LIN {X 0,Y 419.914,Z 1009.254,A -85,B 0,C 180,E1 17766.267,E2 17766.267} C_VEL
LIN {X 0,Y 411.556,Z 1028.718,A -85,B 0,C 180,E1 17763.636,E2 17763.636} C_VEL
LIN {X 0,Y 404.819,Z 1043.815,A -85,B 0,C 180,E1 17761.243,E2 17761.243} C_VEL
LIN {X 0,Y 398.369,Z 1058.063,A -85,B 0,C 180,E1 17758.645,E2 17758.645} C_VEL
LIN {X 0,Y 391.155,Z 1073.748,A -85,B 0,C 180,E1 17755.27,E2 17755.27} C_VEL
LIN {X 0,Y 385.875,Z 1085.364,A -85,B 0,C 180,E1 17752.321,E2 17752.321} C_VEL
LIN {X 0,Y 380.976,Z 1096.633,A -85,B 0,C 180,E1 17748.992,E2 17748.992} C_VEL
LIN {X 0,Y 376.618,Z 1107.153,A -85,B 0,C 180,E1 17745.238,E2 17745.238} C_VEL
LIN {X 0,Y 373.797,Z 1114.641,A -85,B 0,C 180,E1 17742.043,E2 17742.043} C_VEL
LIN {X 0,Y 371.603,Z 1121.269,A -85,B 0,C 180,E1 17738.666,E2 17738.666} C_VEL
LIN {X 0,Y 369.854,Z 1127.751,A -85,B 0,C 180,E1 17734.496,E2 17734.496} C_VEL
LIN {X 0,Y 368.993,Z 1131.833,A -85,B 0,C 180,E1 17730.931,E2 17730.931} C_VEL
LIN {X 0,Y 368.608,Z 1134.428,A -85,B 0,C 180,E1 17727.824,E2 17727.824} C_VEL
LIN {X 0,Y 368.429,Z 1136.13,A -85,B 0,C 180,E1 17724.706,E2 17724.706} C_VEL
LIN {X 0,Y 368.395,Z 1136.967,A -85,B 0,C 180,E1 17721.415,E2 17721.415} C_VEL
LIN {X 0,Y 368.477,Z 1136.697,A -85,B 0,C 180,E1 17717.415,E2 17717.415} C_VEL
LIN {X 0,Y 367.526,Z 1136.369,A -85,B 0,C 180,E1 17716.218,E2 17716.218} C_VEL
LIN {X 0,Y 361.39,Z 1135.259,A -85,B 0,C 180,E1 17712.831,E2 17712.831} C_VEL
LIN {X 0,Y 360.995,Z 1134.749,A -85,B 0,C 180,E1 17711.95,E2 17711.95} C_VEL
LIN {X 0,Y 362,Z 1130.889,A -85,B 0,C 180,E1 17707.716,E2 17707.716} C_VEL
LIN {X 0,Y 363.474,Z 1126.513,A -85,B 0,C 180,E1 17704.238,E2 17704.238} C_VEL
LIN {X 0,Y 365.707,Z 1120.907,A -85,B 0,C 180,E1 17700.699,E2 17700.699} C_VEL
LIN {X 0,Y 369.605,Z 1112.44,A -85,B 0,C 180,E1 17696.432,E2 17696.432} C_VEL
LIN {X 0,Y 374.095,Z 1103.44,A -85,B 0,C 180,E1 17692.798,E2 17692.798} C_VEL
LIN {X 0,Y 379.173,Z 1093.949,A -85,B 0,C 180,E1 17689.557,E2 17689.557} C_VEL
LIN {X 0,Y 386.62,Z 1080.458,A -85,B 0,C 180,E1 17685.712,E2 17685.712} C_VEL
LIN {X 0,Y 393.537,Z 1068.018,A -85,B 0,C 180,E1 17682.755,E2 17682.755} C_VEL
LIN {X 0,Y 400.925,Z 1054.718,A -85,B 0,C 180,E1 17680.038,E2 17680.038} C_VEL
LIN {X 0,Y 410.659,Z 1036.667,A -85,B 0,C 180,E1 17676.93,E2 17676.93} C_VEL
LIN {X 0,Y 418.509,Z 1021.522,A -85,B 0,C 180,E1 17674.73,E2 17674.73} C_VEL
LIN {X 0,Y 426.535,Z 1005.366,A -85,B 0,C 180,E1 17672.696,E2 17672.696} C_VEL
LIN {X 0,Y 436.473,Z 984.02,A -85,B 0,C 180,E1 17670.416,E2 17670.416} C_VEL
LIN {X 0,Y 444.603,Z 964.996,A -85,B 0,C 180,E1 17668.71,E2 17668.71} C_VEL
LIN {X 0,Y 451.802,Z 946.841,A -85,B 0,C 180,E1 17667.31,E2 17667.31} C_VEL
LIN {X 0,Y 459.9,Z 924.448,A -85,B 0,C 180,E1 17665.833,E2 17665.833} C_VEL
LIN {X 0,Y 466.882,Z 902.195,A -85,B 0,C 180,E1 17664.619,E2 17664.619} C_VEL
LIN {X 0,Y 472.272,Z 882.801,A -85,B 0,C 180,E1 17663.72,E2 17663.72} C_VEL
LIN {X 0,Y 477.499,Z 861.186,A -85,B 0,C 180,E1 17662.878,E2 17662.878} C_VEL
LIN {X 0,Y 483.038,Z 832.99,A -85,B 0,C 180,E1 17662.009,E2 17662.009} C_VEL
LIN {X 0,Y 486.435,Z 810.58,A -85,B 0,C 180,E1 17661.488,E2 17661.488} C_VEL
LIN {X 0,Y 488.932,Z 787.935,A -85,B 0,C 180,E1 17661.074,E2 17661.074} C_VEL
LIN {X 0,Y 507.571,Z 549.143,A -85,B 0,C 180,E1 17657.399,E2 17657.399} C_VEL
LIN {X 0,Y 510.985,Z 506.859,A -85,B 0,C 180,E1 17656.756,E2 17656.756} C_VEL
LIN {X 0,Y 505.744,Z 497.944,A -85,B 0,C 180,E1 17654.6,E2 17654.6} C_VEL
LIN {X 0,Y 500.413,Z 489.376,A -85,B 0,C 180,E1 17652.052,E2 17652.052} C_VEL
LIN {X 0,Y 497.211,Z 484.357,A -85,B 0,C 180,E1 17650.252,E2 17650.252} C_VEL
LIN {X 0,Y 494.031,Z 479.444,A -85,B 0,C 180,E1 17648.145,E2 17648.145} C_VEL
LIN {X 0,Y 492.423,Z 477.013,A -85,B 0,C 180,E1 17646.881,E2 17646.881} C_VEL
LIN {X 0,Y 489.648,Z 472.649,A -85,B 0,C 180,E1 17644.099,E2 17644.099} C_VEL
LIN {X 0,Y 487.171,Z 469.067,A -85,B 0,C 180,E1 17638.942,E2 17638.942} C_VEL
LIN {X 0,Y 487.223,Z 469.186,A -85,B 0,C 180,E1 17636.47,E2 17636.47} C_VEL
LIN {X 0,Y 490.053,Z 473.176,A -85,B 0,C 180,E1 17631.138,E2 17631.138} C_VEL
LIN {X 0,Y 493.646,Z 478.878,A -85,B 0,C 180,E1 17627.839,E2 17627.839} C_VEL
LIN {X 0,Y 496.917,Z 484.03,A -85,B 0,C 180,E1 17625.611,E2 17625.611} C_VEL
LIN {X 0,Y 499.764,Z 488.535,A -85,B 0,C 180,E1 17623.972,E2 17623.972} C_VEL
LIN {X 0,Y 504.407,Z 495.808,A -85,B 0,C 180,E1 17621.688,E2 17621.688} C_VEL
LIN {X 0,Y 510.711,Z 506.476,A -85,B 0,C 180,E1 17619.038,E2 17619.038} C_VEL
LIN {X 0,Y 512.388,Z 509.7,A -85,B 0,C 180,E1 17618.385,E2 17618.385} C_VEL
LIN {X 0,Y 495.256,Z 729.15,A -85,B 0,C 180,E1 17614.92,E2 17614.92} C_VEL
LIN {X 0,Y 488.537,Z 815.817,A -85,B 0,C 180,E1 17613.529,E2 17613.529} C_VEL
LIN {X 0,Y 484.757,Z 844.781,A -85,B 0,C 180,E1 17612.964,E2 17612.964} C_VEL
LIN {X 0,Y 480.382,Z 868.6,A -85,B 0,C 180,E1 17612.377,E2 17612.377} C_VEL
LIN {X 0,Y 475.726,Z 889.877,A -85,B 0,C 180,E1 17611.719,E2 17611.719} C_VEL
LIN {X 0,Y 470.261,Z 911.48,A -85,B 0,C 180,E1 17610.91,E2 17610.91} C_VEL
LIN {X 0,Y 462.298,Z 938.776,A -85,B 0,C 180,E1 17609.65,E2 17609.65} C_VEL
LIN {X 0,Y 455.227,Z 960.106,A -85,B 0,C 180,E1 17608.452,E2 17608.452} C_VEL
LIN {X 0,Y 448.224,Z 979.553,A -85,B 0,C 180,E1 17607.174,E2 17607.174} C_VEL
LIN {X 0,Y 440.915,Z 998.4,A -85,B 0,C 180,E1 17605.748,E2 17605.748} C_VEL
LIN {X 0,Y 431.52,Z 1021.146,A -85,B 0,C 180,E1 17603.74,E2 17603.74} C_VEL
LIN {X 0,Y 422.386,Z 1041.626,A -85,B 0,C 180,E1 17601.585,E2 17601.585} C_VEL
LIN {X 0,Y 414.68,Z 1058.316,A -85,B 0,C 180,E1 17599.562,E2 17599.562} C_VEL
LIN {X 0,Y 406.899,Z 1074.752,A -85,B 0,C 180,E1 17597.284,E2 17597.284} C_VEL
LIN {X 0,Y 397.906,Z 1093.613,A -85,B 0,C 180,E1 17594.26,E2 17594.26} C_VEL
LIN {X 0,Y 389.649,Z 1110.63,A -85,B 0,C 180,E1 17591.023,E2 17591.023} C_VEL
LIN {X 0,Y 383.486,Z 1123.697,A -85,B 0,C 180,E1 17588.165,E2 17588.165} C_VEL
LIN {X 0,Y 377.582,Z 1136.795,A -85,B 0,C 180,E1 17584.888,E2 17584.888} C_VEL
LIN {X 0,Y 371.414,Z 1151.399,A -85,B 0,C 180,E1 17580.584,E2 17580.584} C_VEL
LIN {X 0,Y 367.703,Z 1161.191,A -85,B 0,C 180,E1 17577.183,E2 17577.183} C_VEL
LIN {X 0,Y 364.983,Z 1169.338,A -85,B 0,C 180,E1 17573.919,E2 17573.919} C_VEL
LIN {X 0,Y 362.911,Z 1176.713,A -85,B 0,C 180,E1 17570.481,E2 17570.481} C_VEL
LIN {X 0,Y 361.4,Z 1183.466,A -85,B 0,C 180,E1 17566.722,E2 17566.722} C_VEL
LIN {X 0,Y 360.514,Z 1189.451,A -85,B 0,C 180,E1 17562.493,E2 17562.493} C_VEL
LIN {X 0,Y 360.23,Z 1193.242,A -85,B 0,C 180,E1 17558.781,E2 17558.781} C_VEL
LIN {X 0,Y 360.196,Z 1195.573,A -85,B 0,C 180,E1 17555.416,E2 17555.416} C_VEL
LIN {X 0,Y 360.224,Z 1196.781,A -85,B 0,C 180,E1 17552.183,E2 17552.183} C_VEL
LIN {X 0,Y 360.227,Z 1196.963,A -85,B 0,C 180,E1 17549.046,E2 17549.046} C_VEL
LIN {X 0,Y 360.202,Z 1196.137,A -85,B 0,C 180,E1 17545.861,E2 17545.861} C_VEL
LIN {X 0,Y 360.215,Z 1194.293,A -85,B 0,C 180,E1 17542.664,E2 17542.664} C_VEL
LIN {X 0,Y 360.335,Z 1191.418,A -85,B 0,C 180,E1 17539.448,E2 17539.448} C_VEL
LIN {X 0,Y 360.729,Z 1187.502,A -85,B 0,C 180,E1 17536.21,E2 17536.21} C_VEL
LIN {X 0,Y 361.455,Z 1182.799,A -85,B 0,C 180,E1 17533.115,E2 17533.115} C_VEL
LIN {X 0,Y 362.753,Z 1176.781,A -85,B 0,C 180,E1 17529.847,E2 17529.847} C_VEL
LIN {X 0,Y 364.616,Z 1169.625,A -85,B 0,C 180,E1 17526.571,E2 17526.571} C_VEL
LIN {X 0,Y 367.345,Z 1160.858,A -85,B 0,C 180,E1 17523.139,E2 17523.139} C_VEL
LIN {X 0,Y 371.889,Z 1148.059,A -85,B 0,C 180,E1 17518.922,E2 17518.922} C_VEL
LIN {X 0,Y 376.613,Z 1135.964,A -85,B 0,C 180,E1 17515.564,E2 17515.564} C_VEL
LIN {X 0,Y 381.398,Z 1124.305,A -85,B 0,C 180,E1 17512.73,E2 17512.73} C_VEL
LIN {X 0,Y 387.036,Z 1110.995,A -85,B 0,C 180,E1 17509.881,E2 17509.881} C_VEL
LIN {X 0,Y 394.625,Z 1093.507,A -85,B 0,C 180,E1 17506.636,E2 17506.636} C_VEL
LIN {X 0,Y 402.156,Z 1075.877,A -85,B 0,C 180,E1 17503.862,E2 17503.862} C_VEL
LIN {X 0,Y 408.73,Z 1060.305,A -85,B 0,C 180,E1 17501.713,E2 17501.713} C_VEL
LIN {X 0,Y 415.643,Z 1043.455,A -85,B 0,C 180,E1 17499.666,E2 17499.666} C_VEL
LIN {X 0,Y 424.169,Z 1022.004,A -85,B 0,C 180,E1 17497.403,E2 17497.403} C_VEL
LIN {X 0,Y 432.153,Z 1000.246,A -85,B 0,C 180,E1 17495.471,E2 17495.471} C_VEL
LIN {X 0,Y 438.856,Z 980.764,A -85,B 0,C 180,E1 17493.972,E2 17493.972} C_VEL
LIN {X 0,Y 445.267,Z 960.778,A -85,B 0,C 180,E1 17492.641,E2 17492.641} C_VEL
LIN {X 0,Y 452.539,Z 935.959,A -85,B 0,C 180,E1 17491.235,E2 17491.235} C_VEL
LIN {X 0,Y 458.792,Z 911.305,A -85,B 0,C 180,E1 17490.095,E2 17490.095} C_VEL
LIN {X 0,Y 463.496,Z 890.298,A -85,B 0,C 180,E1 17489.286,E2 17489.286} C_VEL
LIN {X 0,Y 467.808,Z 868.068,A -85,B 0,C 180,E1 17488.58,E2 17488.58} C_VEL
LIN {X 0,Y 472.236,Z 839.896,A -85,B 0,C 180,E1 17487.884,E2 17487.884} C_VEL
LIN {X 0,Y 474.871,Z 815.065,A -85,B 0,C 180,E1 17487.405,E2 17487.405} C_VEL
LIN {X 0,Y 488.031,Z 610.604,A -85,B 0,C 180,E1 17484.156,E2 17484.156} C_VEL
LIN {X 0,Y 495.147,Z 501.263,A -85,B 0,C 180,E1 17482.406,E2 17482.406} C_VEL
LIN {X 0,Y 486.329,Z 486.42,A -85,B 0,C 180,E1 17479.956,E2 17479.956} C_VEL
LIN {X 0,Y 478.188,Z 473.236,A -85,B 0,C 180,E1 17477.43,E2 17477.43} C_VEL
LIN {X 0,Y 470.019,Z 460.725,A -85,B 0,C 180,E1 17474.555,E2 17474.555} C_VEL
LIN {X 0,Y 463.191,Z 450.679,A -85,B 0,C 180,E1 17471.771,E2 17471.771} C_VEL
LIN {X 0,Y 459.05,Z 444.945,A -85,B 0,C 180,E1 17469.845,E2 17469.845} C_VEL
LIN {X 0,Y 455.57,Z 439.984,A -85,B 0,C 180,E1 17468.011,E2 17468.011} C_VEL
LIN {X 0,Y 452.275,Z 435.496,A -85,B 0,C 180,E1 17466.028,E2 17466.028} C_VEL
LIN {X 0,Y 449.034,Z 431.044,A -85,B 0,C 180,E1 17463.703,E2 17463.703} C_VEL
LIN {X 0,Y 445.197,Z 425.763,A -85,B 0,C 180,E1 17460,E2 17460} C_VEL
LIN {X 0,Y 442.357,Z 422.52,A -85,B 0,C 180,E1 17454.422,E2 17454.422} C_VEL
LIN {X 0,Y 442.349,Z 422.508,A -85,B 0,C 180,E1 17451.289,E2 17451.289} C_VEL
LIN {X 0,Y 445.229,Z 425.73,A -85,B 0,C 180,E1 17445.565,E2 17445.565} C_VEL
LIN {X 0,Y 449.761,Z 431.958,A -85,B 0,C 180,E1 17441.329,E2 17441.329} C_VEL
LIN {X 0,Y 454.026,Z 437.869,A -85,B 0,C 180,E1 17438.489,E2 17438.489} C_VEL
LIN {X 0,Y 457.249,Z 442.331,A -85,B 0,C 180,E1 17436.684,E2 17436.684} C_VEL
LIN {X 0,Y 461.24,Z 447.999,A -85,B 0,C 180,E1 17434.719,E2 17434.719} C_VEL
LIN {X 0,Y 466.632,Z 455.642,A -85,B 0,C 180,E1 17432.395,E2 17432.395} C_VEL
LIN {X 0,Y 474.915,Z 468.281,A -85,B 0,C 180,E1 17429.299,E2 17429.299} C_VEL
LIN {X 0,Y 483.221,Z 481.644,A -85,B 0,C 180,E1 17426.604,E2 17426.604} C_VEL
LIN {X 0,Y 491.26,Z 495.152,A -85,B 0,C 180,E1 17424.279,E2 17424.279} C_VEL
LIN {X 0,Y 476.265,Z 720.31,A -85,B 0,C 180,E1 17420.785,E2 17420.785} C_VEL
LIN {X 0,Y 471.261,Z 794.313,A -85,B 0,C 180,E1 17419.609,E2 17419.609} C_VEL
LIN {X 0,Y 467.909,Z 823.069,A -85,B 0,C 180,E1 17418.995,E2 17418.995} C_VEL
LIN {X 0,Y 464.464,Z 844.981,A -85,B 0,C 180,E1 17418.365,E2 17418.365} C_VEL
LIN {X 0,Y 460.75,Z 864.458,A -85,B 0,C 180,E1 17417.684,E2 17417.684} C_VEL
LIN {X 0,Y 455.503,Z 888.033,A -85,B 0,C 180,E1 17416.691,E2 17416.691} C_VEL
LIN {X 0,Y 449.095,Z 912.163,A -85,B 0,C 180,E1 17415.434,E2 17415.434} C_VEL
LIN {X 0,Y 443.4,Z 931.244,A -85,B 0,C 180,E1 17414.26,E2 17414.26} C_VEL
LIN {X 0,Y 436.845,Z 951.268,A -85,B 0,C 180,E1 17412.826,E2 17412.826} C_VEL
LIN {X 0,Y 428.599,Z 973.995,A -85,B 0,C 180,E1 17410.898,E2 17410.898} C_VEL
LIN {X 0,Y 421.57,Z 991.841,A -85,B 0,C 180,E1 17409.115,E2 17409.115} C_VEL
LIN {X 0,Y 414.534,Z 1008.746,A -85,B 0,C 180,E1 17407.172,E2 17407.172} C_VEL
LIN {X 0,Y 405.844,Z 1028.465,A -85,B 0,C 180,E1 17404.516,E2 17404.516} C_VEL
LIN {X 0,Y 398.838,Z 1043.639,A -85,B 0,C 180,E1 17402.105,E2 17402.105} C_VEL
LIN {X 0,Y 392.449,Z 1057.236,A -85,B 0,C 180,E1 17399.621,E2 17399.621} C_VEL
LIN {X 0,Y 385.195,Z 1072.591,A -85,B 0,C 180,E1 17396.351,E2 17396.351} C_VEL
LIN {X 0,Y 379.154,Z 1085.231,A -85,B 0,C 180,E1 17393.136,E2 17393.136} C_VEL
LIN {X 0,Y 374.507,Z 1095.344,A -85,B 0,C 180,E1 17390.145,E2 17390.145} C_VEL
LIN {X 0,Y 369.769,Z 1106.289,A -85,B 0,C 180,E1 17386.333,E2 17386.333} C_VEL
LIN {X 0,Y 366.269,Z 1114.954,A -85,B 0,C 180,E1 17382.614,E2 17382.614} C_VEL
LIN {X 0,Y 364.005,Z 1121.345,A -85,B 0,C 180,E1 17379.327,E2 17379.327} C_VEL
LIN {X 0,Y 362.247,Z 1127.354,A -85,B 0,C 180,E1 17375.544,E2 17375.544} C_VEL
LIN {X 0,Y 361.11,Z 1132.183,A -85,B 0,C 180,E1 17371.428,E2 17371.428} C_VEL
LIN {X 0,Y 360.665,Z 1134.97,A -85,B 0,C 180,E1 17368.093,E2 17368.093} C_VEL
LIN {X 0,Y 360.464,Z 1136.716,A -85,B 0,C 180,E1 17364.908,E2 17364.908} C_VEL
LIN {X 0,Y 360.426,Z 1137.574,A -85,B 0,C 180,E1 17361.706,E2 17361.706} C_VEL
LIN {X 0,Y 360.467,Z 1137.524,A -85,B 0,C 180,E1 17358.289,E2 17358.289} C_VEL
LIN {X 0,Y 360.722,Z 1136.104,A -85,B 0,C 180,E1 17354.125,E2 17354.125} C_VEL
LIN {X 0,Y 360.995,Z 1134.749,A -85,B 0,C 180,E1 17351.95,E2 17351.95} C_VEL
LIN {X 0,Y 360.233,Z 1133.997,A -85,B 0,C 180,E1 17350.729,E2 17350.729} C_VEL
LIN {X 0,Y 354.802,Z 1131.503,A -85,B 0,C 180,E1 17347.361,E2 17347.361} C_VEL
LIN {X 0,Y 354.533,Z 1130.483,A -85,B 0,C 180,E1 17346.384,E2 17346.384} C_VEL
LIN {X 0,Y 356.672,Z 1125.074,A -85,B 0,C 180,E1 17342.267,E2 17342.267} C_VEL
LIN {X 0,Y 359.898,Z 1117.871,A -85,B 0,C 180,E1 17338.139,E2 17338.139} C_VEL
LIN {X 0,Y 363.572,Z 1110.604,A -85,B 0,C 180,E1 17334.724,E2 17334.724} C_VEL
LIN {X 0,Y 368.537,Z 1101.516,A -85,B 0,C 180,E1 17331.139,E2 17331.139} C_VEL
LIN {X 0,Y 375.404,Z 1089.408,A -85,B 0,C 180,E1 17327.221,E2 17327.221} C_VEL
LIN {X 0,Y 381.927,Z 1078.151,A -85,B 0,C 180,E1 17324.167,E2 17324.167} C_VEL
LIN {X 0,Y 389.377,Z 1065.395,A -85,B 0,C 180,E1 17321.203,E2 17321.203} C_VEL
LIN {X 0,Y 398.644,Z 1049.164,A -85,B 0,C 180,E1 17318.042,E2 17318.042} C_VEL
LIN {X 0,Y 406.699,Z 1034.589,A -85,B 0,C 180,E1 17315.639,E2 17315.639} C_VEL
LIN {X 0,Y 415.054,Z 1018.938,A -85,B 0,C 180,E1 17313.414,E2 17313.414} C_VEL
LIN {X 0,Y 425.458,Z 998.249,A -85,B 0,C 180,E1 17310.932,E2 17310.932} C_VEL
LIN {X 0,Y 433.487,Z 981.035,A -85,B 0,C 180,E1 17309.187,E2 17309.187} C_VEL
LIN {X 0,Y 441.247,Z 963.214,A -85,B 0,C 180,E1 17307.625,E2 17307.625} C_VEL
LIN {X 0,Y 449.982,Z 941.493,A -85,B 0,C 180,E1 17305.999,E2 17305.999} C_VEL
LIN {X 0,Y 457.976,Z 918.744,A -85,B 0,C 180,E1 17304.59,E2 17304.59} C_VEL
LIN {X 0,Y 464.159,Z 899.184,A -85,B 0,C 180,E1 17303.569,E2 17303.569} C_VEL
LIN {X 0,Y 469.902,Z 878.59,A -85,B 0,C 180,E1 17302.653,E2 17302.653} C_VEL
LIN {X 0,Y 476.01,Z 852.496,A -85,B 0,C 180,E1 17301.707,E2 17301.707} C_VEL
LIN {X 0,Y 480.18,Z 830.257,A -85,B 0,C 180,E1 17301.065,E2 17301.065} C_VEL
LIN {X 0,Y 483.513,Z 808.071,A -85,B 0,C 180,E1 17300.567,E2 17300.567} C_VEL
LIN {X 0,Y 486.548,Z 778.332,A -85,B 0,C 180,E1 17300.055,E2 17300.055} C_VEL
LIN {X 0,Y 505.512,Z 541.034,A -85,B 0,C 180,E1 17296.42,E2 17296.42} C_VEL
LIN {X 0,Y 507.889,Z 512.008,A -85,B 0,C 180,E1 17295.97,E2 17295.97} C_VEL
LIN {X 0,Y 503.019,Z 503.688,A -85,B 0,C 180,E1 17293.859,E2 17293.859} C_VEL
LIN {X 0,Y 498.361,Z 496.107,A -85,B 0,C 180,E1 17291.516,E2 17291.516} C_VEL
LIN {X 0,Y 495.476,Z 491.467,A -85,B 0,C 180,E1 17289.818,E2 17289.818} C_VEL
LIN {X 0,Y 491.73,Z 485.38,A -85,B 0,C 180,E1 17287.125,E2 17287.125} C_VEL
LIN {X 0,Y 488.568,Z 480.528,A -85,B 0,C 180,E1 17283.99,E2 17283.99} C_VEL
LIN {X 0,Y 486.191,Z 477.013,A -85,B 0,C 180,E1 17278.939,E2 17278.939} C_VEL
LIN {X 0,Y 486.223,Z 477.089,A -85,B 0,C 180,E1 17276.581,E2 17276.581} C_VEL
LIN {X 0,Y 488.918,Z 480.985,A -85,B 0,C 180,E1 17271.295,E2 17271.295} C_VEL
LIN {X 0,Y 492.427,Z 486.698,A -85,B 0,C 180,E1 17267.987,E2 17267.987} C_VEL
LIN {X 0,Y 495.646,Z 491.876,A -85,B 0,C 180,E1 17265.752,E2 17265.752} C_VEL
LIN {X 0,Y 498.45,Z 496.423,A -85,B 0,C 180,E1 17264.108,E2 17264.108} C_VEL
LIN {X 0,Y 502.954,Z 503.677,A -85,B 0,C 180,E1 17261.851,E2 17261.851} C_VEL
LIN {X 0,Y 508.789,Z 513.771,A -85,B 0,C 180,E1 17259.344,E2 17259.344} C_VEL
LIN {X 0,Y 509.234,Z 514.927,A -85,B 0,C 180,E1 17259.152,E2 17259.152} C_VEL
LIN {X 0,Y 491.623,Z 734.941,A -85,B 0,C 180,E1 17255.685,E2 17255.685} C_VEL
LIN {X 0,Y 485.171,Z 815.707,A -85,B 0,C 180,E1 17254.388,E2 17254.388} C_VEL
LIN {X 0,Y 481.157,Z 845.436,A -85,B 0,C 180,E1 17253.808,E2 17253.808} C_VEL
LIN {X 0,Y 476.817,Z 868.51,A -85,B 0,C 180,E1 17253.243,E2 17253.243} C_VEL
LIN {X 0,Y 472.149,Z 889.384,A -85,B 0,C 180,E1 17252.603,E2 17252.603} C_VEL
LIN {X 0,Y 466.733,Z 910.328,A -85,B 0,C 180,E1 17251.828,E2 17251.828} C_VEL
LIN {X 0,Y 459.059,Z 936.319,A -85,B 0,C 180,E1 17250.654,E2 17250.654} C_VEL
LIN {X 0,Y 451.328,Z 959.125,A -85,B 0,C 180,E1 17249.392,E2 17249.392} C_VEL
LIN {X 0,Y 444.324,Z 978.128,A -85,B 0,C 180,E1 17248.156,E2 17248.156} C_VEL
LIN {X 0,Y 436.91,Z 996.727,A -85,B 0,C 180,E1 17246.766,E2 17246.766} C_VEL
LIN {X 0,Y 427.495,Z 1018.957,A -85,B 0,C 180,E1 17244.829,E2 17244.829} C_VEL
LIN {X 0,Y 417.765,Z 1040.189,A -85,B 0,C 180,E1 17242.617,E2 17242.617} C_VEL
LIN {X 0,Y 409.438,Z 1057.619,A -85,B 0,C 180,E1 17240.505,E2 17240.505} C_VEL
LIN {X 0,Y 401.441,Z 1073.901,A -85,B 0,C 180,E1 17238.241,E2 17238.241} C_VEL
LIN {X 0,Y 391.983,Z 1092.974,A -85,B 0,C 180,E1 17235.163,E2 17235.163} C_VEL
LIN {X 0,Y 383.74,Z 1109.281,A -85,B 0,C 180,E1 17232.039,E2 17232.039} C_VEL
LIN {X 0,Y 376.875,Z 1123.132,A -85,B 0,C 180,E1 17228.98,E2 17228.98} C_VEL
LIN {X 0,Y 370.629,Z 1136.272,A -85,B 0,C 180,E1 17225.641,E2 17225.641} C_VEL
LIN {X 0,Y 364.314,Z 1150.44,A -85,B 0,C 180,E1 17221.398,E2 17221.398} C_VEL
LIN {X 0,Y 360.227,Z 1160.611,A -85,B 0,C 180,E1 17217.795,E2 17217.795} C_VEL
LIN {X 0,Y 357.216,Z 1169.126,A -85,B 0,C 180,E1 17214.297,E2 17214.297} C_VEL
LIN {X 0,Y 354.954,Z 1176.759,A -85,B 0,C 180,E1 17210.616,E2 17210.616} C_VEL
LIN {X 0,Y 353.234,Z 1184.407,A -85,B 0,C 180,E1 17206.105,E2 17206.105} C_VEL
LIN {X 0,Y 352.477,Z 1189.527,A -85,B 0,C 180,E1 17202.117,E2 17202.117} C_VEL
LIN {X 0,Y 352.247,Z 1192.729,A -85,B 0,C 180,E1 17198.817,E2 17198.817} C_VEL
LIN {X 0,Y 352.216,Z 1194.927,A -85,B 0,C 180,E1 17195.539,E2 17195.539} C_VEL
LIN {X 0,Y 352.249,Z 1196.119,A -85,B 0,C 180,E1 17192.278,E2 17192.278} C_VEL
LIN {X 0,Y 352.254,Z 1196.298,A -85,B 0,C 180,E1 17189.024,E2 17189.024} C_VEL
LIN {X 0,Y 352.228,Z 1195.531,A -85,B 0,C 180,E1 17185.931,E2 17185.931} C_VEL
LIN {X 0,Y 352.235,Z 1193.719,A -85,B 0,C 180,E1 17182.661,E2 17182.661} C_VEL
LIN {X 0,Y 352.353,Z 1190.875,A -85,B 0,C 180,E1 17179.371,E2 17179.371} C_VEL
LIN {X 0,Y 352.761,Z 1186.987,A -85,B 0,C 180,E1 17176.059,E2 17176.059} C_VEL
LIN {X 0,Y 353.574,Z 1182.029,A -85,B 0,C 180,E1 17172.727,E2 17172.727} C_VEL
LIN {X 0,Y 354.953,Z 1175.979,A -85,B 0,C 180,E1 17169.384,E2 17169.384} C_VEL
LIN {X 0,Y 357.024,Z 1168.54,A -85,B 0,C 180,E1 17165.925,E2 17165.925} C_VEL
LIN {X 0,Y 360.489,Z 1158.228,A -85,B 0,C 180,E1 17161.868,E2 17161.868} C_VEL
LIN {X 0,Y 365.072,Z 1146.011,A -85,B 0,C 180,E1 17157.905,E2 17157.905} C_VEL
LIN {X 0,Y 369.636,Z 1134.842,A -85,B 0,C 180,E1 17154.779,E2 17154.779} C_VEL
LIN {X 0,Y 374.898,Z 1122.588,A -85,B 0,C 180,E1 17151.775,E2 17151.775} C_VEL
LIN {X 0,Y 382.118,Z 1106.477,A -85,B 0,C 180,E1 17148.347,E2 17148.347} C_VEL
LIN {X 0,Y 389.996,Z 1088.705,A -85,B 0,C 180,E1 17145.168,E2 17145.168} C_VEL
LIN {X 0,Y 396.677,Z 1073.642,A -85,B 0,C 180,E1 17142.82,E2 17142.82} C_VEL
LIN {X 0,Y 403.671,Z 1057.583,A -85,B 0,C 180,E1 17140.62,E2 17140.62} C_VEL
LIN {X 0,Y 412.505,Z 1036.71,A -85,B 0,C 180,E1 17138.136,E2 17138.136} C_VEL
LIN {X 0,Y 420.851,Z 1015.583,A -85,B 0,C 180,E1 17136.022,E2 17136.022} C_VEL
LIN {X 0,Y 427.822,Z 997.015,A -85,B 0,C 180,E1 17134.413,E2 17134.413} C_VEL
LIN {X 0,Y 434.45,Z 978.156,A -85,B 0,C 180,E1 17132.984,E2 17132.984} C_VEL
LIN {X 0,Y 442.411,Z 953.671,A -85,B 0,C 180,E1 17131.395,E2 17131.395} C_VEL
LIN {X 0,Y 449.242,Z 929.745,A -85,B 0,C 180,E1 17130.119,E2 17130.119} C_VEL
LIN {X 0,Y 454.619,Z 908.745,A -85,B 0,C 180,E1 17129.175,E2 17129.175} C_VEL
LIN {X 0,Y 459.575,Z 886.857,A -85,B 0,C 180,E1 17128.354,E2 17128.354} C_VEL
LIN {X 0,Y 464.799,Z 859.411,A -85,B 0,C 180,E1 17127.527,E2 17127.527} C_VEL
LIN {X 0,Y 468.468,Z 834.345,A -85,B 0,C 180,E1 17126.958,E2 17126.958} C_VEL
LIN {X 0,Y 470.749,Z 811.97,A -85,B 0,C 180,E1 17126.536,E2 17126.536} C_VEL
LIN {X 0,Y 484.922,Z 597.377,A -85,B 0,C 180,E1 17123.126,E2 17123.126} C_VEL
LIN {X 0,Y 491.073,Z 505.694,A -85,B 0,C 180,E1 17121.66,E2 17121.66} C_VEL
LIN {X 0,Y 481.939,Z 490.181,A -85,B 0,C 180,E1 17119.01,E2 17119.01} C_VEL
LIN {X 0,Y 474.495,Z 478.138,A -85,B 0,C 180,E1 17116.591,E2 17116.591} C_VEL
LIN {X 0,Y 467.344,Z 466.91,A -85,B 0,C 180,E1 17113.959,E2 17113.959} C_VEL
LIN {X 0,Y 460.815,Z 457.299,A -85,B 0,C 180,E1 17111.198,E2 17111.198} C_VEL
LIN {X 0,Y 457.297,Z 452.287,A -85,B 0,C 180,E1 17109.502,E2 17109.502} C_VEL
LIN {X 0,Y 454.005,Z 447.502,A -85,B 0,C 180,E1 17107.721,E2 17107.721} C_VEL
LIN {X 0,Y 450.787,Z 443.042,A -85,B 0,C 180,E1 17105.729,E2 17105.729} C_VEL
LIN {X 0,Y 447.711,Z 438.746,A -85,B 0,C 180,E1 17103.457,E2 17103.457} C_VEL
LIN {X 0,Y 444.103,Z 433.636,A -85,B 0,C 180,E1 17099.871,E2 17099.871} C_VEL
LIN {X 0,Y 441.377,Z 430.463,A -85,B 0,C 180,E1 17094.41,E2 17094.41} C_VEL
LIN {X 0,Y 441.355,Z 430.423,A -85,B 0,C 180,E1 17091.401,E2 17091.401} C_VEL
LIN {X 0,Y 443.95,Z 433.452,A -85,B 0,C 180,E1 17085.922,E2 17085.922} C_VEL
LIN {X 0,Y 444.804,Z 434.715,A -85,B 0,C 180,E1 17084.885,E2 17084.885} C_VEL
LIN {X 0,Y 448.551,Z 439.817,A -85,B 0,C 180,E1 17081.479,E2 17081.479} C_VEL
LIN {X 0,Y 452.758,Z 445.742,A -85,B 0,C 180,E1 17078.63,E2 17078.63} C_VEL
LIN {X 0,Y 455.824,Z 450.09,A -85,B 0,C 180,E1 17076.88,E2 17076.88} C_VEL
LIN {X 0,Y 459.76,Z 455.78,A -85,B 0,C 180,E1 17074.907,E2 17074.907} C_VEL
LIN {X 0,Y 464.893,Z 463.214,A -85,B 0,C 180,E1 17072.654,E2 17072.654} C_VEL
LIN {X 0,Y 472.793,Z 475.492,A -85,B 0,C 180,E1 17069.636,E2 17069.636} C_VEL
LIN {X 0,Y 480.783,Z 488.57,A -85,B 0,C 180,E1 17066.983,E2 17066.983} C_VEL
LIN {X 0,Y 487.267,Z 499.765,A -85,B 0,C 180,E1 17065.041,E2 17065.041} C_VEL
LIN {X 0,Y 471.335,Z 732.845,A -85,B 0,C 180,E1 17061.422,E2 17061.422} C_VEL
LIN {X 0,Y 466.938,Z 795.404,A -85,B 0,C 180,E1 17060.423,E2 17060.423} C_VEL
LIN {X 0,Y 463.508,Z 823.863,A -85,B 0,C 180,E1 17059.812,E2 17059.812} C_VEL
LIN {X 0,Y 460.001,Z 845.637,A -85,B 0,C 180,E1 17059.184,E2 17059.184} C_VEL
LIN {X 0,Y 456.202,Z 865.097,A -85,B 0,C 180,E1 17058.505,E2 17058.505} C_VEL
LIN {X 0,Y 450.555,Z 889.852,A -85,B 0,C 180,E1 17057.456,E2 17057.456} C_VEL
LIN {X 0,Y 443.992,Z 913.723,A -85,B 0,C 180,E1 17056.2,E2 17056.2} C_VEL
LIN {X 0,Y 438.164,Z 932.693,A -85,B 0,C 180,E1 17055.023,E2 17055.023} C_VEL
LIN {X 0,Y 430.665,Z 954.936,A -85,B 0,C 180,E1 17053.41,E2 17053.41} C_VEL
LIN {X 0,Y 422.409,Z 976.679,A -85,B 0,C 180,E1 17051.511,E2 17051.511} C_VEL
LIN {X 0,Y 415.54,Z 993.596,A -85,B 0,C 180,E1 17049.795,E2 17049.795} C_VEL
LIN {X 0,Y 407.268,Z 1012.863,A -85,B 0,C 180,E1 17047.533,E2 17047.533} C_VEL
LIN {X 0,Y 398.971,Z 1030.81,A -85,B 0,C 180,E1 17045.022,E2 17045.022} C_VEL
LIN {X 0,Y 392.185,Z 1045.047,A -85,B 0,C 180,E1 17042.716,E2 17042.716} C_VEL
LIN {X 0,Y 385.262,Z 1059.302,A -85,B 0,C 180,E1 17040.059,E2 17040.059} C_VEL
LIN {X 0,Y 377.498,Z 1074.994,A -85,B 0,C 180,E1 17036.591,E2 17036.591} C_VEL
LIN {X 0,Y 371.874,Z 1086.394,A -85,B 0,C 180,E1 17033.617,E2 17033.617} C_VEL
LIN {X 0,Y 366.847,Z 1096.937,A -85,B 0,C 180,E1 17030.418,E2 17030.418} C_VEL
LIN {X 0,Y 361.63,Z 1108.425,A -85,B 0,C 180,E1 17026.215,E2 17026.215} C_VEL
LIN {X 0,Y 358.512,Z 1115.918,A -85,B 0,C 180,E1 17022.892,E2 17022.892} C_VEL
LIN {X 0,Y 356.067,Z 1122.549,A -85,B 0,C 180,E1 17019.373,E2 17019.373} C_VEL
LIN {X 0,Y 354.101,Z 1129.036,A -85,B 0,C 180,E1 17015.022,E2 17015.022} C_VEL
LIN {X 0,Y 353.124,Z 1133.121,A -85,B 0,C 180,E1 17011.298,E2 17011.298} C_VEL
LIN {X 0,Y 352.691,Z 1135.721,A -85,B 0,C 180,E1 17008.05,E2 17008.05} C_VEL
LIN {X 0,Y 352.487,Z 1137.431,A -85,B 0,C 180,E1 17004.792,E2 17004.792} C_VEL
LIN {X 0,Y 352.449,Z 1138.254,A -85,B 0,C 180,E1 17001.517,E2 17001.517} C_VEL
LIN {X 0,Y 352.525,Z 1138.142,A -85,B 0,C 180,E1 16997.718,E2 16997.718} C_VEL
LIN {X 0,Y 352.817,Z 1136.546,A -85,B 0,C 180,E1 16993.537,E2 16993.537} C_VEL
LIN {X 0,Y 353.431,Z 1134.014,A -85,B 0,C 180,E1 16989.929,E2 16989.929} C_VEL
LIN {X 0,Y 354.533,Z 1130.483,A -85,B 0,C 180,E1 16986.384,E2 16986.384} C_VEL
LIN {X 0,Y 354.088,Z 1129.241,A -85,B 0,C 180,E1 16985.148,E2 16985.148} C_VEL
LIN {X 0,Y 349.723,Z 1125.58,A -85,B 0,C 180,E1 16981.716,E2 16981.716} C_VEL
LIN {X 0,Y 349.774,Z 1124.115,A -85,B 0,C 180,E1 16980.741,E2 16980.741} C_VEL
LIN {X 0,Y 352.993,Z 1117.602,A -85,B 0,C 180,E1 16977.054,E2 16977.054} C_VEL
LIN {X 0,Y 357.487,Z 1109.408,A -85,B 0,C 180,E1 16973.235,E2 16973.235} C_VEL
LIN {X 0,Y 363.852,Z 1098.416,A -85,B 0,C 180,E1 16969.089,E2 16969.089} C_VEL
LIN {X 0,Y 370.116,Z 1087.968,A -85,B 0,C 180,E1 16965.815,E2 16965.815} C_VEL
LIN {X 0,Y 377.928,Z 1075.22,A -85,B 0,C 180,E1 16962.428,E2 16962.428} C_VEL
LIN {X 0,Y 386.853,Z 1060.348,A -85,B 0,C 180,E1 16959.161,E2 16959.161} C_VEL
LIN {X 0,Y 394.883,Z 1046.7,A -85,B 0,C 180,E1 16956.616,E2 16956.616} C_VEL
LIN {X 0,Y 403.604,Z 1031.43,A -85,B 0,C 180,E1 16954.165,E2 16954.165} C_VEL
LIN {X 0,Y 414.115,Z 1011.928,A -85,B 0,C 180,E1 16951.537,E2 16951.537} C_VEL
LIN {X 0,Y 422.542,Z 995.275,A -85,B 0,C 180,E1 16949.642,E2 16949.642} C_VEL
LIN {X 0,Y 430.598,Z 978.338,A -85,B 0,C 180,E1 16947.974,E2 16947.974} C_VEL
LIN {X 0,Y 440.157,Z 956.588,A -85,B 0,C 180,E1 16946.149,E2 16946.149} C_VEL
LIN {X 0,Y 448.392,Z 935.532,A -85,B 0,C 180,E1 16944.677,E2 16944.677} C_VEL
LIN {X 0,Y 455.259,Z 916.132,A -85,B 0,C 180,E1 16943.518,E2 16943.518} C_VEL
LIN {X 0,Y 462.673,Z 892.73,A -85,B 0,C 180,E1 16942.342,E2 16942.342} C_VEL
LIN {X 0,Y 469.125,Z 868.23,A -85,B 0,C 180,E1 16941.348,E2 16941.348} C_VEL
LIN {X 0,Y 473.754,Z 847.581,A -85,B 0,C 180,E1 16940.664,E2 16940.664} C_VEL
LIN {X 0,Y 477.642,Z 826.548,A -85,B 0,C 180,E1 16940.089,E2 16940.089} C_VEL
LIN {X 0,Y 481.564,Z 798.45,A -85,B 0,C 180,E1 16939.508,E2 16939.508} C_VEL
LIN {X 0,Y 486.408,Z 741.305,A -85,B 0,C 180,E1 16938.61,E2 16938.61} C_VEL
LIN {X 0,Y 504.933,Z 517.336,A -85,B 0,C 180,E1 16935.197,E2 16935.197} C_VEL
LIN {X 0,Y 500.267,Z 509.262,A -85,B 0,C 180,E1 16933.053,E2 16933.053} C_VEL
LIN {X 0,Y 495.322,Z 500.924,A -85,B 0,C 180,E1 16930.35,E2 16930.35} C_VEL
LIN {X 0,Y 491.296,Z 494.541,A -85,B 0,C 180,E1 16927.602,E2 16927.602} C_VEL
LIN {X 0,Y 489.644,Z 492.084,A -85,B 0,C 180,E1 16926.213,E2 16926.213} C_VEL
LIN {X 0,Y 487.492,Z 488.407,A -85,B 0,C 180,E1 16923.881,E2 16923.881} C_VEL
LIN {X 0,Y 485.198,Z 484.919,A -85,B 0,C 180,E1 16918.819,E2 16918.819} C_VEL
LIN {X 0,Y 485.259,Z 485.091,A -85,B 0,C 180,E1 16916.456,E2 16916.456} C_VEL
LIN {X 0,Y 487.876,Z 489.008,A -85,B 0,C 180,E1 16911.336,E2 16911.336} C_VEL
LIN {X 0,Y 491.141,Z 494.393,A -85,B 0,C 180,E1 16908.194,E2 16908.194} C_VEL
LIN {X 0,Y 494.29,Z 499.575,A -85,B 0,C 180,E1 16905.951,E2 16905.951} C_VEL
LIN {X 0,Y 497.14,Z 504.306,A -85,B 0,C 180,E1 16904.245,E2 16904.245} C_VEL
LIN {X 0,Y 501.657,Z 511.808,A -85,B 0,C 180,E1 16901.944,E2 16901.944} C_VEL
LIN {X 0,Y 506.195,Z 519.849,A -85,B 0,C 180,E1 16899.935,E2 16899.935} C_VEL
LIN {X 0,Y 488.485,Z 735.729,A -85,B 0,C 180,E1 16896.541,E2 16896.541} C_VEL
LIN {X 0,Y 481.963,Z 815.229,A -85,B 0,C 180,E1 16895.267,E2 16895.267} C_VEL
LIN {X 0,Y 477.92,Z 844.694,A -85,B 0,C 180,E1 16894.696,E2 16894.696} C_VEL
LIN {X 0,Y 473.42,Z 868.148,A -85,B 0,C 180,E1 16894.128,E2 16894.128} C_VEL
LIN {X 0,Y 468.722,Z 888.75,A -85,B 0,C 180,E1 16893.504,E2 16893.504} C_VEL
LIN {X 0,Y 462.981,Z 910.483,A -85,B 0,C 180,E1 16892.708,E2 16892.708} C_VEL
LIN {X 0,Y 454.68,Z 937.651,A -85,B 0,C 180,E1 16891.477,E2 16891.477} C_VEL
LIN {X 0,Y 447.08,Z 959.445,A -85,B 0,C 180,E1 16890.269,E2 16890.269} C_VEL
LIN {X 0,Y 439.726,Z 978.823,A -85,B 0,C 180,E1 16889.007,E2 16889.007} C_VEL
LIN {X 0,Y 431.519,Z 998.787,A -85,B 0,C 180,E1 16887.502,E2 16887.502} C_VEL
LIN {X 0,Y 420.712,Z 1023.093,A -85,B 0,C 180,E1 16885.316,E2 16885.316} C_VEL
LIN {X 0,Y 412.185,Z 1041.027,A -85,B 0,C 180,E1 16883.41,E2 16883.41} C_VEL
LIN {X 0,Y 403.883,Z 1057.806,A -85,B 0,C 180,E1 16881.357,E2 16881.357} C_VEL
LIN {X 0,Y 394.891,Z 1075.477,A -85,B 0,C 180,E1 16878.863,E2 16878.863} C_VEL
LIN {X 0,Y 384.758,Z 1094.935,A -85,B 0,C 180,E1 16875.613,E2 16875.613} C_VEL
LIN {X 0,Y 377.039,Z 1109.655,A -85,B 0,C 180,E1 16872.727,E2 16872.727} C_VEL
LIN {X 0,Y 370.277,Z 1122.719,A -85,B 0,C 180,E1 16869.79,E2 16869.79} C_VEL
LIN {X 0,Y 363.193,Z 1136.965,A -85,B 0,C 180,E1 16866.096,E2 16866.096} C_VEL
LIN {X 0,Y 356.814,Z 1150.526,A -85,B 0,C 180,E1 16861.887,E2 16861.887} C_VEL
LIN {X 0,Y 352.613,Z 1160.475,A -85,B 0,C 180,E1 16858.264,E2 16858.264} C_VEL
LIN {X 0,Y 349.461,Z 1168.918,A -85,B 0,C 180,E1 16854.691,E2 16854.691} C_VEL
LIN {X 0,Y 346.748,Z 1177.794,A -85,B 0,C 180,E1 16850.244,E2 16850.244} C_VEL
LIN {X 0,Y 345.152,Z 1184.694,A -85,B 0,C 180,E1 16845.802,E2 16845.802} C_VEL
LIN {X 0,Y 344.496,Z 1189.075,A -85,B 0,C 180,E1 16842.232,E2 16842.232} C_VEL
LIN {X 0,Y 344.263,Z 1192.22,A -85,B 0,C 180,E1 16838.855,E2 16838.855} C_VEL
LIN {X 0,Y 344.234,Z 1194.283,A -85,B 0,C 180,E1 16835.668,E2 16835.668} C_VEL
LIN {X 0,Y 344.275,Z 1195.466,A -85,B 0,C 180,E1 16832.33,E2 16832.33} C_VEL
LIN {X 0,Y 344.279,Z 1195.656,A -85,B 0,C 180,E1 16829.168,E2 16829.168} C_VEL
LIN {X 0,Y 344.254,Z 1194.852,A -85,B 0,C 180,E1 16825.836,E2 16825.836} C_VEL
LIN {X 0,Y 344.256,Z 1193.021,A -85,B 0,C 180,E1 16822.49,E2 16822.49} C_VEL
LIN {X 0,Y 344.381,Z 1190.152,A -85,B 0,C 180,E1 16819.122,E2 16819.122} C_VEL
LIN {X 0,Y 344.829,Z 1186.238,A -85,B 0,C 180,E1 16815.732,E2 16815.732} C_VEL
LIN {X 0,Y 345.708,Z 1181.255,A -85,B 0,C 180,E1 16812.321,E2 16812.321} C_VEL
LIN {X 0,Y 347.168,Z 1175.172,A -85,B 0,C 180,E1 16808.9,E2 16808.9} C_VEL
LIN {X 0,Y 349.429,Z 1167.568,A -85,B 0,C 180,E1 16805.307,E2 16805.307} C_VEL
LIN {X 0,Y 353.27,Z 1156.705,A -85,B 0,C 180,E1 16800.997,E2 16800.997} C_VEL
LIN {X 0,Y 357.889,Z 1145.056,A -85,B 0,C 180,E1 16797.181,E2 16797.181} C_VEL
LIN {X 0,Y 362.614,Z 1133.979,A -85,B 0,C 180,E1 16794.033,E2 16794.033} C_VEL
LIN {X 0,Y 368.202,Z 1121.546,A -85,B 0,C 180,E1 16790.95,E2 16790.95} C_VEL
LIN {X 0,Y 375.744,Z 1105.354,A -85,B 0,C 180,E1 16787.476,E2 16787.476} C_VEL
LIN {X 0,Y 383.523,Z 1088.411,A -85,B 0,C 180,E1 16784.412,E2 16784.412} C_VEL
LIN {X 0,Y 390.647,Z 1072.873,A -85,B 0,C 180,E1 16781.967,E2 16781.967} C_VEL
LIN {X 0,Y 398.393,Z 1055.667,A -85,B 0,C 180,E1 16779.603,E2 16779.603} C_VEL
LIN {X 0,Y 408.288,Z 1032.63,A -85,B 0,C 180,E1 16776.911,E2 16776.911} C_VEL
LIN {X 0,Y 415.807,Z 1014.152,A -85,B 0,C 180,E1 16775.08,E2 16775.08} C_VEL
LIN {X 0,Y 423.053,Z 995.341,A -85,B 0,C 180,E1 16773.458,E2 16773.458} C_VEL
LIN {X 0,Y 430.202,Z 975.468,A -85,B 0,C 180,E1 16771.971,E2 16771.971} C_VEL
LIN {X 0,Y 438.576,Z 949.755,A -85,B 0,C 180,E1 16770.346,E2 16770.346} C_VEL
LIN {X 0,Y 444.857,Z 928.184,A -85,B 0,C 180,E1 16769.215,E2 16769.215} C_VEL
LIN {X 0,Y 450.406,Z 906.864,A -85,B 0,C 180,E1 16768.268,E2 16768.268} C_VEL
LIN {X 0,Y 456.168,Z 881.67,A -85,B 0,C 180,E1 16767.346,E2 16767.346} C_VEL
LIN {X 0,Y 461.087,Z 854.939,A -85,B 0,C 180,E1 16766.591,E2 16766.591} C_VEL
LIN {X 0,Y 464.364,Z 832.381,A -85,B 0,C 180,E1 16766.09,E2 16766.09} C_VEL
LIN {X 0,Y 466.688,Z 809.289,A -85,B 0,C 180,E1 16765.66,E2 16765.66} C_VEL
LIN {X 0,Y 481.583,Z 589.499,A -85,B 0,C 180,E1 16762.169,E2 16762.169} C_VEL
LIN {X 0,Y 487.066,Z 510.157,A -85,B 0,C 180,E1 16760.9,E2 16760.9} C_VEL
LIN {X 0,Y 477.764,Z 494.125,A -85,B 0,C 180,E1 16758.075,E2 16758.075} C_VEL
LIN {X 0,Y 470.12,Z 481.714,A -85,B 0,C 180,E1 16755.45,E2 16755.45} C_VEL
LIN {X 0,Y 462.908,Z 470.36,A -85,B 0,C 180,E1 16752.601,E2 16752.601} C_VEL
LIN {X 0,Y 456.649,Z 461.03,A -85,B 0,C 180,E1 16749.707,E2 16749.707} C_VEL
LIN {X 0,Y 452.239,Z 454.739,A -85,B 0,C 180,E1 16747.304,E2 16747.304} C_VEL
LIN {X 0,Y 449.404,Z 450.701,A -85,B 0,C 180,E1 16745.49,E2 16745.49} C_VEL
LIN {X 0,Y 446.556,Z 446.608,A -85,B 0,C 180,E1 16743.337,E2 16743.337} C_VEL
LIN {X 0,Y 443.01,Z 441.508,A -85,B 0,C 180,E1 16739.741,E2 16739.741} C_VEL
LIN {X 0,Y 440.396,Z 438.405,A -85,B 0,C 180,E1 16734.397,E2 16734.397} C_VEL
LIN {X 0,Y 440.38,Z 438.373,A -85,B 0,C 180,E1 16731.381,E2 16731.381} C_VEL
LIN {X 0,Y 443.216,Z 441.608,A -85,B 0,C 180,E1 16725.631,E2 16725.631} C_VEL
LIN {X 0,Y 446.716,Z 446.681,A -85,B 0,C 180,E1 16722.142,E2 16722.142} C_VEL
LIN {X 0,Y 451.29,Z 453.319,A -85,B 0,C 180,E1 16718.897,E2 16718.897} C_VEL
LIN {X 0,Y 454.292,Z 457.669,A -85,B 0,C 180,E1 16717.14,E2 16717.14} C_VEL
LIN {X 0,Y 458.031,Z 463.179,A -85,B 0,C 180,E1 16715.22,E2 16715.22} C_VEL
LIN {X 0,Y 463.19,Z 470.829,A -85,B 0,C 180,E1 16712.904,E2 16712.904} C_VEL
LIN {X 0,Y 470.676,Z 482.683,A -85,B 0,C 180,E1 16709.981,E2 16709.981} C_VEL
LIN {X 0,Y 478.366,Z 495.495,A -85,B 0,C 180,E1 16707.365,E2 16707.365} C_VEL
LIN {X 0,Y 483.349,Z 504.367,A -85,B 0,C 180,E1 16705.818,E2 16705.818} C_VEL
LIN {X 0,Y 466.873,Z 739.32,A -85,B 0,C 180,E1 16702.168,E2 16702.168} C_VEL
LIN {X 0,Y 462.729,Z 796.29,A -85,B 0,C 180,E1 16701.255,E2 16701.255} C_VEL
LIN {X 0,Y 459.23,Z 824.482,A -85,B 0,C 180,E1 16700.648,E2 16700.648} C_VEL
LIN {X 0,Y 455.672,Z 846.078,A -85,B 0,C 180,E1 16700.026,E2 16700.026} C_VEL
LIN {X 0,Y 451.747,Z 865.715,A -85,B 0,C 180,E1 16699.342,E2 16699.342} C_VEL
LIN {X 0,Y 445.968,Z 890.436,A -85,B 0,C 180,E1 16698.295,E2 16698.295} C_VEL
LIN {X 0,Y 439.541,Z 913.35,A -85,B 0,C 180,E1 16697.094,E2 16697.094} C_VEL
LIN {X 0,Y 433.471,Z 932.722,A -85,B 0,C 180,E1 16695.899,E2 16695.899} C_VEL
LIN {X 0,Y 426.407,Z 953.216,A -85,B 0,C 180,E1 16694.422,E2 16694.422} C_VEL
LIN {X 0,Y 417.642,Z 975.992,A -85,B 0,C 180,E1 16692.464,E2 16692.464} C_VEL
LIN {X 0,Y 410.309,Z 993.6,A -85,B 0,C 180,E1 16690.681,E2 16690.681} C_VEL
LIN {X 0,Y 402.634,Z 1010.991,A -85,B 0,C 180,E1 16688.649,E2 16688.649} C_VEL
LIN {X 0,Y 393.417,Z 1030.535,A -85,B 0,C 180,E1 16685.95,E2 16685.95} C_VEL
LIN {X 0,Y 386.367,Z 1044.852,A -85,B 0,C 180,E1 16683.628,E2 16683.628} C_VEL
LIN {X 0,Y 379.515,Z 1058.463,A -85,B 0,C 180,E1 16681.089,E2 16681.089} C_VEL
LIN {X 0,Y 371.701,Z 1073.826,A -85,B 0,C 180,E1 16677.733,E2 16677.733} C_VEL
LIN {X 0,Y 365.166,Z 1086.475,A -85,B 0,C 180,E1 16674.422,E2 16674.422} C_VEL
LIN {X 0,Y 360.092,Z 1096.599,A -85,B 0,C 180,E1 16671.33,E2 16671.33} C_VEL
LIN {X 0,Y 354.906,Z 1107.552,A -85,B 0,C 180,E1 16667.375,E2 16667.375} C_VEL
LIN {X 0,Y 351.037,Z 1116.222,A -85,B 0,C 180,E1 16663.507,E2 16663.507} C_VEL
LIN {X 0,Y 348.523,Z 1122.618,A -85,B 0,C 180,E1 16660.079,E2 16660.079} C_VEL
LIN {X 0,Y 346.479,Z 1128.869,A -85,B 0,C 180,E1 16655.963,E2 16655.963} C_VEL
LIN {X 0,Y 345.252,Z 1133.469,A -85,B 0,C 180,E1 16651.825,E2 16651.825} C_VEL
LIN {X 0,Y 344.75,Z 1136.26,A -85,B 0,C 180,E1 16648.338,E2 16648.338} C_VEL
LIN {X 0,Y 344.521,Z 1138.015,A -85,B 0,C 180,E1 16645.005,E2 16645.005} C_VEL
LIN {X 0,Y 344.477,Z 1138.886,A -85,B 0,C 180,E1 16641.655,E2 16641.655} C_VEL
LIN {X 0,Y 344.532,Z 1138.855,A -85,B 0,C 180,E1 16638.109,E2 16638.109} C_VEL
LIN {X 0,Y 344.83,Z 1137.538,A -85,B 0,C 180,E1 16633.838,E2 16633.838} C_VEL
LIN {X 0,Y 345.493,Z 1134.903,A -85,B 0,C 180,E1 16629.856,E2 16629.856} C_VEL
LIN {X 0,Y 346.662,Z 1131.394,A -85,B 0,C 180,E1 16626.184,E2 16626.184} C_VEL
LIN {X 0,Y 348.621,Z 1126.634,A -85,B 0,C 180,E1 16622.407,E2 16622.407} C_VEL
LIN {X 0,Y 349.774,Z 1124.115,A -85,B 0,C 180,E1 16620.741,E2 16620.741} C_VEL
LIN {X 0,Y 349.751,Z 1122.291,A -85,B 0,C 180,E1 16619.507,E2 16619.507} C_VEL
LIN {X 0,Y 346.718,Z 1117.427,A -85,B 0,C 180,E1 16616.043,E2 16616.043} C_VEL
LIN {X 0,Y 347.173,Z 1115.712,A -85,B 0,C 180,E1 16615.075,E2 16615.075} C_VEL
LIN {X 0,Y 352.708,Z 1106.26,A -85,B 0,C 180,E1 16610.965,E2 16610.965} C_VEL
LIN {X 0,Y 358.248,Z 1097.291,A -85,B 0,C 180,E1 16607.7,E2 16607.7} C_VEL
LIN {X 0,Y 365.45,Z 1085.967,A -85,B 0,C 180,E1 16604.207,E2 16604.207} C_VEL
LIN {X 0,Y 374.274,Z 1072.009,A -85,B 0,C 180,E1 16600.651,E2 16600.651} C_VEL
LIN {X 0,Y 382.419,Z 1058.938,A -85,B 0,C 180,E1 16597.852,E2 16597.852} C_VEL
LIN {X 0,Y 390.847,Z 1045.094,A -85,B 0,C 180,E1 16595.308,E2 16595.308} C_VEL
LIN {X 0,Y 401.633,Z 1026.553,A -85,B 0,C 180,E1 16592.442,E2 16592.442} C_VEL
LIN {X 0,Y 410.606,Z 1010.173,A -85,B 0,C 180,E1 16590.318,E2 16590.318} C_VEL
LIN {X 0,Y 419.018,Z 993.952,A -85,B 0,C 180,E1 16588.506,E2 16588.506} C_VEL
LIN {X 0,Y 428.63,Z 974.156,A -85,B 0,C 180,E1 16586.608,E2 16586.608} C_VEL
LIN {X 0,Y 438.087,Z 952.375,A -85,B 0,C 180,E1 16584.875,E2 16584.875} C_VEL
LIN {X 0,Y 445.314,Z 934.178,A -85,B 0,C 180,E1 16583.641,E2 16583.641} C_VEL
LIN {X 0,Y 452.719,Z 913.545,A -85,B 0,C 180,E1 16582.439,E2 16582.439} C_VEL
LIN {X 0,Y 460.66,Z 888.018,A -85,B 0,C 180,E1 16581.216,E2 16581.216} C_VEL
LIN {X 0,Y 466.349,Z 866.45,A -85,B 0,C 180,E1 16580.369,E2 16580.369} C_VEL
LIN {X 0,Y 471.248,Z 844.635,A -85,B 0,C 180,E1 16579.67,E2 16579.67} C_VEL
LIN {X 0,Y 475.966,Z 818.172,A -85,B 0,C 180,E1 16579.003,E2 16579.003} C_VEL
LIN {X 0,Y 478.966,Z 794.473,A -85,B 0,C 180,E1 16578.552,E2 16578.552} C_VEL
LIN {X 0,Y 498.3,Z 565.958,A -85,B 0,C 180,E1 16575.058,E2 16575.058} C_VEL
LIN {X 0,Y 502.012,Z 522.56,A -85,B 0,C 180,E1 16574.387,E2 16574.387} C_VEL
LIN {X 0,Y 496.467,Z 512.909,A -85,B 0,C 180,E1 16571.619,E2 16571.619} C_VEL
LIN {X 0,Y 492.685,Z 506.682,A -85,B 0,C 180,E1 16569.344,E2 16569.344} C_VEL
LIN {X 0,Y 489.335,Z 500.973,A -85,B 0,C 180,E1 16566.806,E2 16566.806} C_VEL
LIN {X 0,Y 486.325,Z 496.196,A -85,B 0,C 180,E1 16563.654,E2 16563.654} C_VEL
LIN {X 0,Y 484.218,Z 492.864,A -85,B 0,C 180,E1 16558.817,E2 16558.817} C_VEL
LIN {X 0,Y 484.277,Z 493.046,A -85,B 0,C 180,E1 16556.449,E2 16556.449} C_VEL
LIN {X 0,Y 486.79,Z 496.922,A -85,B 0,C 180,E1 16551.436,E2 16551.436} C_VEL
LIN {X 0,Y 489.933,Z 502.212,A -85,B 0,C 180,E1 16548.343,E2 16548.343} C_VEL
LIN {X 0,Y 493.027,Z 507.419,A -85,B 0,C 180,E1 16546.094,E2 16546.094} C_VEL
LIN {X 0,Y 496.869,Z 513.82,A -85,B 0,C 180,E1 16543.816,E2 16543.816} C_VEL
LIN {X 0,Y 501.651,Z 522.234,A -85,B 0,C 180,E1 16541.433,E2 16541.433} C_VEL
LIN {X 0,Y 503.228,Z 525.236,A -85,B 0,C 180,E1 16540.716,E2 16540.716} C_VEL
LIN {X 0,Y 484.802,Z 744.578,A -85,B 0,C 180,E1 16537.28,E2 16537.28} C_VEL
LIN {X 0,Y 478.816,Z 815.339,A -85,B 0,C 180,E1 16536.147,E2 16536.147} C_VEL
LIN {X 0,Y 474.541,Z 845.425,A -85,B 0,C 180,E1 16535.564,E2 16535.564} C_VEL
LIN {X 0,Y 470.078,Z 868.147,A -85,B 0,C 180,E1 16535.018,E2 16535.018} C_VEL
LIN {X 0,Y 465.159,Z 889.178,A -85,B 0,C 180,E1 16534.385,E2 16534.385} C_VEL
LIN {X 0,Y 458.982,Z 911.927,A -85,B 0,C 180,E1 16533.551,E2 16533.551} C_VEL
LIN {X 0,Y 450.473,Z 938.772,A -85,B 0,C 180,E1 16532.327,E2 16532.327} C_VEL
LIN {X 0,Y 443.235,Z 959.017,A -85,B 0,C 180,E1 16531.209,E2 16531.209} C_VEL
LIN {X 0,Y 435.944,Z 977.761,A -85,B 0,C 180,E1 16529.999,E2 16529.999} C_VEL
LIN {X 0,Y 427.766,Z 997.144,A -85,B 0,C 180,E1 16528.556,E2 16528.556} C_VEL
LIN {X 0,Y 417.233,Z 1020.395,A -85,B 0,C 180,E1 16526.506,E2 16526.506} C_VEL
LIN {X 0,Y 407.721,Z 1039.808,A -85,B 0,C 180,E1 16524.464,E2 16524.464} C_VEL
LIN {X 0,Y 398.956,Z 1056.97,A -85,B 0,C 180,E1 16522.369,E2 16522.369} C_VEL
LIN {X 0,Y 390.158,Z 1073.654,A -85,B 0,C 180,E1 16520.018,E2 16520.018} C_VEL
LIN {X 0,Y 379.314,Z 1093.725,A -85,B 0,C 180,E1 16516.679,E2 16516.679} C_VEL
LIN {X 0,Y 371.296,Z 1108.38,A -85,B 0,C 180,E1 16513.794,E2 16513.794} C_VEL
LIN {X 0,Y 364.141,Z 1121.584,A -85,B 0,C 180,E1 16510.806,E2 16510.806} C_VEL
LIN {X 0,Y 357.557,Z 1134.063,A -85,B 0,C 180,E1 16507.561,E2 16507.561} C_VEL
LIN {X 0,Y 350.251,Z 1148.777,A -85,B 0,C 180,E1 16503.042,E2 16503.042} C_VEL
LIN {X 0,Y 345.561,Z 1159.047,A -85,B 0,C 180,E1 16499.274,E2 16499.274} C_VEL
LIN {X 0,Y 342.131,Z 1167.582,A -85,B 0,C 180,E1 16495.628,E2 16495.628} C_VEL
LIN {X 0,Y 339.503,Z 1175.239,A -85,B 0,C 180,E1 16491.782,E2 16491.782} C_VEL
LIN {X 0,Y 337.525,Z 1182.707,A -85,B 0,C 180,E1 16487.232,E2 16487.232} C_VEL
LIN {X 0,Y 336.576,Z 1188.092,A -85,B 0,C 180,E1 16482.874,E2 16482.874} C_VEL
LIN {X 0,Y 336.289,Z 1191.457,A -85,B 0,C 180,E1 16479.239,E2 16479.239} C_VEL
LIN {X 0,Y 336.251,Z 1193.561,A -85,B 0,C 180,E1 16475.974,E2 16475.974} C_VEL
LIN {X 0,Y 336.298,Z 1194.786,A -85,B 0,C 180,E1 16472.551,E2 16472.551} C_VEL
LIN {X 0,Y 336.307,Z 1194.99,A -85,B 0,C 180,E1 16469.148,E2 16469.148} C_VEL
LIN {X 0,Y 336.279,Z 1194.243,A -85,B 0,C 180,E1 16465.908,E2 16465.908} C_VEL
LIN {X 0,Y 336.276,Z 1192.442,A -85,B 0,C 180,E1 16462.483,E2 16462.483} C_VEL
LIN {X 0,Y 336.4,Z 1189.602,A -85,B 0,C 180,E1 16459.034,E2 16459.034} C_VEL
LIN {X 0,Y 336.866,Z 1185.714,A -85,B 0,C 180,E1 16455.563,E2 16455.563} C_VEL
LIN {X 0,Y 337.786,Z 1180.751,A -85,B 0,C 180,E1 16452.071,E2 16452.071} C_VEL
LIN {X 0,Y 339.31,Z 1174.689,A -85,B 0,C 180,E1 16448.568,E2 16448.568} C_VEL
LIN {X 0,Y 341.547,Z 1167.493,A -85,B 0,C 180,E1 16445.068,E2 16445.068} C_VEL
LIN {X 0,Y 345.115,Z 1157.734,A -85,B 0,C 180,E1 16441.043,E2 16441.043} C_VEL
LIN {X 0,Y 350.292,Z 1145.185,A -85,B 0,C 180,E1 16436.758,E2 16436.758} C_VEL
LIN {X 0,Y 355.436,Z 1133.592,A -85,B 0,C 180,E1 16433.39,E2 16433.39} C_VEL
LIN {X 0,Y 361.09,Z 1121.52,A -85,B 0,C 180,E1 16430.337,E2 16430.337} C_VEL
LIN {X 0,Y 368.691,Z 1105.798,A -85,B 0,C 180,E1 16426.89,E2 16426.89} C_VEL
LIN {X 0,Y 377.115,Z 1088.107,A -85,B 0,C 180,E1 16423.63,E2 16423.63} C_VEL
LIN {X 0,Y 384.707,Z 1072.103,A -85,B 0,C 180,E1 16421.087,E2 16421.087} C_VEL
LIN {X 0,Y 392.713,Z 1054.865,A -85,B 0,C 180,E1 16418.707,E2 16418.707} C_VEL
LIN {X 0,Y 402.924,Z 1031.786,A -85,B 0,C 180,E1 16416.005,E2 16416.005} C_VEL
LIN {X 0,Y 410.761,Z 1013.027,A -85,B 0,C 180,E1 16414.146,E2 16414.146} C_VEL
LIN {X 0,Y 418.04,Z 994.588,A -85,B 0,C 180,E1 16412.559,E2 16412.559} C_VEL
LIN {X 0,Y 425.983,Z 973.056,A -85,B 0,C 180,E1 16410.959,E2 16410.959} C_VEL
LIN {X 0,Y 434.006,Z 948.786,A -85,B 0,C 180,E1 16409.445,E2 16409.445} C_VEL
LIN {X 0,Y 440.353,Z 927.436,A -85,B 0,C 180,E1 16408.331,E2 16408.331} C_VEL
LIN {X 0,Y 445.798,Z 906.974,A -85,B 0,C 180,E1 16407.426,E2 16407.426} C_VEL
LIN {X 0,Y 451.276,Z 883.618,A -85,B 0,C 180,E1 16406.568,E2 16406.568} C_VEL
LIN {X 0,Y 456.671,Z 855.516,A -85,B 0,C 180,E1 16405.761,E2 16405.761} C_VEL
LIN {X 0,Y 460.112,Z 832.432,A -85,B 0,C 180,E1 16405.248,E2 16405.248} C_VEL
LIN {X 0,Y 462.476,Z 809.636,A -85,B 0,C 180,E1 16404.822,E2 16404.822} C_VEL
LIN {X 0,Y 477.663,Z 591.643,A -85,B 0,C 180,E1 16401.356,E2 16401.356} C_VEL
LIN {X 0,Y 483.137,Z 514.577,A -85,B 0,C 180,E1 16400.125,E2 16400.125} C_VEL
LIN {X 0,Y 473.858,Z 498.506,A -85,B 0,C 180,E1 16397.182,E2 16397.182} C_VEL
LIN {X 0,Y 465.757,Z 485.172,A -85,B 0,C 180,E1 16394.23,E2 16394.23} C_VEL
LIN {X 0,Y 458.303,Z 473.438,A -85,B 0,C 180,E1 16391.037,E2 16391.037} C_VEL
LIN {X 0,Y 453.716,Z 466.798,A -85,B 0,C 180,E1 16388.746,E2 16388.746} C_VEL
LIN {X 0,Y 450.806,Z 462.392,A -85,B 0,C 180,E1 16387.071,E2 16387.071} C_VEL
LIN {X 0,Y 447.938,Z 458.243,A -85,B 0,C 180,E1 16385.187,E2 16385.187} C_VEL
LIN {X 0,Y 445.245,Z 454.309,A -85,B 0,C 180,E1 16383.09,E2 16383.09} C_VEL
LIN {X 0,Y 441.916,Z 449.38,A -85,B 0,C 180,E1 16379.611,E2 16379.611} C_VEL
LIN {X 0,Y 439.396,Z 446.305,A -85,B 0,C 180,E1 16374.254,E2 16374.254} C_VEL
LIN {X 0,Y 439.424,Z 446.366,A -85,B 0,C 180,E1 16371.231,E2 16371.231} C_VEL
LIN {X 0,Y 442.202,Z 449.611,A -85,B 0,C 180,E1 16365.665,E2 16365.665} C_VEL
LIN {X 0,Y 446.064,Z 455.399,A -85,B 0,C 180,E1 16361.845,E2 16361.845} C_VEL
LIN {X 0,Y 450.131,Z 461.335,A -85,B 0,C 180,E1 16358.977,E2 16358.977} C_VEL
LIN {X 0,Y 452.994,Z 465.598,A -85,B 0,C 180,E1 16357.277,E2 16357.277} C_VEL
LIN {X 0,Y 458.06,Z 473.038,A -85,B 0,C 180,E1 16354.704,E2 16354.704} C_VEL
LIN {X 0,Y 464.26,Z 482.909,A -85,B 0,C 180,E1 16351.997,E2 16351.997} C_VEL
LIN {X 0,Y 471.181,Z 494.249,A -85,B 0,C 180,E1 16349.382,E2 16349.382} C_VEL
LIN {X 0,Y 477.834,Z 505.725,A -85,B 0,C 180,E1 16347.146,E2 16347.146} C_VEL
LIN {X 0,Y 479.52,Z 508.895,A -85,B 0,C 180,E1 16346.608,E2 16346.608} C_VEL
LIN {X 0,Y 462.641,Z 743.514,A -85,B 0,C 180,E1 16342.964,E2 16342.964} C_VEL
LIN {X 0,Y 458.607,Z 797.208,A -85,B 0,C 180,E1 16342.101,E2 16342.101} C_VEL
LIN {X 0,Y 455.058,Z 825.023,A -85,B 0,C 180,E1 16341.501,E2 16341.501} C_VEL
LIN {X 0,Y 451.449,Z 846.466,A -85,B 0,C 180,E1 16340.886,E2 16340.886} C_VEL
LIN {X 0,Y 447.391,Z 866.333,A -85,B 0,C 180,E1 16340.195,E2 16340.195} C_VEL
LIN {X 0,Y 441.479,Z 891.018,A -85,B 0,C 180,E1 16339.151,E2 16339.151} C_VEL
LIN {X 0,Y 434.905,Z 913.921,A -85,B 0,C 180,E1 16337.952,E2 16337.952} C_VEL
LIN {X 0,Y 428.797,Z 932.977,A -85,B 0,C 180,E1 16336.777,E2 16336.777} C_VEL
LIN {X 0,Y 422.011,Z 952.243,A -85,B 0,C 180,E1 16335.395,E2 16335.395} C_VEL
LIN {X 0,Y 412.807,Z 975.76,A -85,B 0,C 180,E1 16333.393,E2 16333.393} C_VEL
LIN {X 0,Y 405.182,Z 993.603,A -85,B 0,C 180,E1 16331.59,E2 16331.59} C_VEL
LIN {X 0,Y 397.506,Z 1010.522,A -85,B 0,C 180,E1 16329.616,E2 16329.616} C_VEL
LIN {X 0,Y 387.976,Z 1030.25,A -85,B 0,C 180,E1 16326.903,E2 16326.903} C_VEL
LIN {X 0,Y 380.243,Z 1045.453,A -85,B 0,C 180,E1 16324.426,E2 16324.426} C_VEL
LIN {X 0,Y 373.064,Z 1059.229,A -85,B 0,C 180,E1 16321.828,E2 16321.828} C_VEL
LIN {X 0,Y 364.705,Z 1075.029,A -85,B 0,C 180,E1 16318.313,E2 16318.313} C_VEL
LIN {X 0,Y 358.246,Z 1087.094,A -85,B 0,C 180,E1 16315.102,E2 16315.102} C_VEL
LIN {X 0,Y 352.947,Z 1097.221,A -85,B 0,C 180,E1 16311.959,E2 16311.959} C_VEL
LIN {X 0,Y 347.52,Z 1108.174,A -85,B 0,C 180,E1 16307.93,E2 16307.93} C_VEL
LIN {X 0,Y 343.453,Z 1116.853,A -85,B 0,C 180,E1 16303.983,E2 16303.983} C_VEL
LIN {X 0,Y 340.805,Z 1123.252,A -85,B 0,C 180,E1 16300.48,E2 16300.48} C_VEL
LIN {X 0,Y 338.636,Z 1129.504,A -85,B 0,C 180,E1 16296.272,E2 16296.272} C_VEL
LIN {X 0,Y 337.329,Z 1134.108,A -85,B 0,C 180,E1 16292.038,E2 16292.038} C_VEL
LIN {X 0,Y 336.794,Z 1136.903,A -85,B 0,C 180,E1 16288.469,E2 16288.469} C_VEL
LIN {X 0,Y 336.55,Z 1138.663,A -85,B 0,C 180,E1 16285.057,E2 16285.057} C_VEL
LIN {X 0,Y 336.503,Z 1139.541,A -85,B 0,C 180,E1 16281.628,E2 16281.628} C_VEL
LIN {X 0,Y 336.557,Z 1139.535,A -85,B 0,C 180,E1 16278.171,E2 16278.171} C_VEL
LIN {X 0,Y 336.826,Z 1138.445,A -85,B 0,C 180,E1 16274.117,E2 16274.117} C_VEL
LIN {X 0,Y 337.568,Z 1135.746,A -85,B 0,C 180,E1 16269.724,E2 16269.724} C_VEL
LIN {X 0,Y 338.801,Z 1132.296,A -85,B 0,C 180,E1 16265.967,E2 16265.967} C_VEL
LIN {X 0,Y 340.682,Z 1127.958,A -85,B 0,C 180,E1 16262.373,E2 16262.373} C_VEL
LIN {X 0,Y 344.042,Z 1121.383,A -85,B 0,C 180,E1 16258.065,E2 16258.065} C_VEL
LIN {X 0,Y 347.173,Z 1115.712,A -85,B 0,C 180,E1 16255.075,E2 16255.075} C_VEL
LIN {X 0,Y 347.675,Z 1113.494,A -85,B 0,C 180,E1 16253.85,E2 16253.85} C_VEL
LIN {X 0,Y 346.118,Z 1107.442,A -85,B 0,C 180,E1 16250.494,E2 16250.494} C_VEL
LIN {X 0,Y 346.995,Z 1105.104,A -85,B 0,C 180,E1 16249.473,E2 16249.473} C_VEL
LIN {X 0,Y 354.636,Z 1093.572,A -85,B 0,C 180,E1 16245.41,E2 16245.41} C_VEL
LIN {X 0,Y 362.855,Z 1081.047,A -85,B 0,C 180,E1 16241.826,E2 16241.826} C_VEL
LIN {X 0,Y 370.705,Z 1069.133,A -85,B 0,C 180,E1 16238.937,E2 16238.937} C_VEL
LIN {X 0,Y 380.739,Z 1053.64,A -85,B 0,C 180,E1 16235.761,E2 16235.761} C_VEL
LIN {X 0,Y 390.535,Z 1037.64,A -85,B 0,C 180,E1 16233.048,E2 16233.048} C_VEL
LIN {X 0,Y 399.464,Z 1022.461,A -85,B 0,C 180,E1 16230.848,E2 16230.848} C_VEL
LIN {X 0,Y 409.817,Z 1003.952,A -85,B 0,C 180,E1 16228.56,E2 16228.56} C_VEL
LIN {X 0,Y 420.068,Z 983.824,A -85,B 0,C 180,E1 16226.496,E2 16226.496} C_VEL
LIN {X 0,Y 428.421,Z 966.144,A -85,B 0,C 180,E1 16224.948,E2 16224.948} C_VEL
LIN {X 0,Y 437.422,Z 945.439,A -85,B 0,C 180,E1 16223.401,E2 16223.401} C_VEL
LIN {X 0,Y 446.327,Z 922.231,A -85,B 0,C 180,E1 16221.961,E2 16221.961} C_VEL
LIN {X 0,Y 453.439,Z 901.275,A -85,B 0,C 180,E1 16220.879,E2 16220.879} C_VEL
LIN {X 0,Y 459.685,Z 880.353,A -85,B 0,C 180,E1 16219.968,E2 16219.968} C_VEL
LIN {X 0,Y 466.199,Z 854.342,A -85,B 0,C 180,E1 16219.046,E2 16219.046} C_VEL
LIN {X 0,Y 470.687,Z 831.913,A -85,B 0,C 180,E1 16218.412,E2 16218.412} C_VEL
LIN {X 0,Y 474.218,Z 809.858,A -85,B 0,C 180,E1 16217.927,E2 16217.927} C_VEL
LIN {X 0,Y 477.359,Z 781.739,A -85,B 0,C 180,E1 16217.446,E2 16217.446} C_VEL
LIN {X 0,Y 497.841,Z 543.967,A -85,B 0,C 180,E1 16213.844,E2 16213.844} C_VEL
LIN {X 0,Y 499.213,Z 528.007,A -85,B 0,C 180,E1 16213.585,E2 16213.585} C_VEL
LIN {X 0,Y 494.053,Z 519.016,A -85,B 0,C 180,E1 16210.849,E2 16210.849} C_VEL
LIN {X 0,Y 490.459,Z 512.72,A -85,B 0,C 180,E1 16208.5,E2 16208.5} C_VEL
LIN {X 0,Y 487.805,Z 508.356,A -85,B 0,C 180,E1 16206.355,E2 16206.355} C_VEL
LIN {X 0,Y 485.255,Z 504.076,A -85,B 0,C 180,E1 16203.544,E2 16203.544} C_VEL
LIN {X 0,Y 483.227,Z 500.772,A -85,B 0,C 180,E1 16198.696,E2 16198.696} C_VEL
LIN {X 0,Y 483.295,Z 501.001,A -85,B 0,C 180,E1 16196.442,E2 16196.442} C_VEL
LIN {X 0,Y 485.705,Z 504.835,A -85,B 0,C 180,E1 16191.536,E2 16191.536} C_VEL
LIN {X 0,Y 488.722,Z 510.019,A -85,B 0,C 180,E1 16188.499,E2 16188.499} C_VEL
LIN {X 0,Y 491.854,Z 515.402,A -85,B 0,C 180,E1 16186.18,E2 16186.18} C_VEL
LIN {X 0,Y 496.059,Z 522.724,A -85,B 0,C 180,E1 16183.669,E2 16183.669} C_VEL
LIN {X 0,Y 500.373,Z 530.443,A -85,B 0,C 180,E1 16181.512,E2 16181.512} C_VEL
LIN {X 0,Y 481.573,Z 749.083,A -85,B 0,C 180,E1 16178.1,E2 16178.1} C_VEL
LIN {X 0,Y 475.812,Z 815.23,A -85,B 0,C 180,E1 16177.043,E2 16177.043} C_VEL
LIN {X 0,Y 471.49,Z 844.996,A -85,B 0,C 180,E1 16176.469,E2 16176.469} C_VEL
LIN {X 0,Y 466.946,Z 867.717,A -85,B 0,C 180,E1 16175.93,E2 16175.93} C_VEL
LIN {X 0,Y 461.923,Z 888.777,A -85,B 0,C 180,E1 16175.306,E2 16175.306} C_VEL
LIN {X 0,Y 455.451,Z 912.13,A -85,B 0,C 180,E1 16174.459,E2 16174.459} C_VEL
LIN {X 0,Y 446.979,Z 938.2,A -85,B 0,C 180,E1 16173.279,E2 16173.279} C_VEL
LIN {X 0,Y 439.364,Z 958.979,A -85,B 0,C 180,E1 16172.142,E2 16172.142} C_VEL
LIN {X 0,Y 431.571,Z 978.474,A -85,B 0,C 180,E1 16170.886,E2 16170.886} C_VEL
LIN {X 0,Y 421.596,Z 1001.452,A -85,B 0,C 180,E1 16169.151,E2 16169.151} C_VEL
LIN {X 0,Y 411.153,Z 1023.259,A -85,B 0,C 180,E1 16167.158,E2 16167.158} C_VEL
LIN {X 0,Y 402.175,Z 1040.986,A -85,B 0,C 180,E1 16165.264,E2 16165.264} C_VEL
LIN {X 0,Y 393.337,Z 1057.696,A -85,B 0,C 180,E1 16163.2,E2 16163.2} C_VEL
LIN {X 0,Y 382.722,Z 1077.167,A -85,B 0,C 180,E1 16160.396,E2 16160.396} C_VEL
LIN {X 0,Y 372.63,Z 1094.908,A -85,B 0,C 180,E1 16157.325,E2 16157.325} C_VEL
LIN {X 0,Y 364.741,Z 1108.766,A -85,B 0,C 180,E1 16154.54,E2 16154.54} C_VEL
LIN {X 0,Y 357.38,Z 1121.781,A -85,B 0,C 180,E1 16151.534,E2 16151.534} C_VEL
LIN {X 0,Y 349.196,Z 1136.732,A -85,B 0,C 180,E1 16147.517,E2 16147.517} C_VEL
LIN {X 0,Y 342.424,Z 1149.698,A -85,B 0,C 180,E1 16143.295,E2 16143.295} C_VEL
LIN {X 0,Y 338.018,Z 1158.925,A -85,B 0,C 180,E1 16139.798,E2 16139.798} C_VEL
LIN {X 0,Y 334.424,Z 1167.387,A -85,B 0,C 180,E1 16136.072,E2 16136.072} C_VEL
LIN {X 0,Y 331.371,Z 1175.962,A -85,B 0,C 180,E1 16131.599,E2 16131.599} C_VEL
LIN {X 0,Y 329.431,Z 1183.006,A -85,B 0,C 180,E1 16126.94,E2 16126.94} C_VEL
LIN {X 0,Y 328.623,Z 1187.479,A -85,B 0,C 180,E1 16123.18,E2 16123.18} C_VEL
LIN {X 0,Y 328.313,Z 1190.825,A -85,B 0,C 180,E1 16119.466,E2 16119.466} C_VEL
LIN {X 0,Y 328.271,Z 1192.919,A -85,B 0,C 180,E1 16116.12,E2 16116.12} C_VEL
LIN {X 0,Y 328.322,Z 1194.133,A -85,B 0,C 180,E1 16112.618,E2 16112.618} C_VEL
LIN {X 0,Y 328.332,Z 1194.347,A -85,B 0,C 180,E1 16109.302,E2 16109.302} C_VEL
LIN {X 0,Y 328.304,Z 1193.56,A -85,B 0,C 180,E1 16105.808,E2 16105.808} C_VEL
LIN {X 0,Y 328.296,Z 1191.738,A -85,B 0,C 180,E1 16102.299,E2 16102.299} C_VEL
LIN {X 0,Y 328.433,Z 1188.873,A -85,B 0,C 180,E1 16098.765,E2 16098.765} C_VEL
LIN {X 0,Y 328.953,Z 1184.885,A -85,B 0,C 180,E1 16095.151,E2 16095.151} C_VEL
LIN {X 0,Y 329.955,Z 1179.82,A -85,B 0,C 180,E1 16091.534,E2 16091.534} C_VEL
LIN {X 0,Y 331.559,Z 1173.871,A -85,B 0,C 180,E1 16088.041,E2 16088.041} C_VEL
LIN {X 0,Y 334.09,Z 1166.233,A -85,B 0,C 180,E1 16084.272,E2 16084.272} C_VEL
LIN {X 0,Y 338.283,Z 1155.516,A -85,B 0,C 180,E1 16079.837,E2 16079.837} C_VEL
LIN {X 0,Y 343.476,Z 1143.543,A -85,B 0,C 180,E1 16075.767,E2 16075.767} C_VEL
LIN {X 0,Y 348.608,Z 1132.585,A -85,B 0,C 180,E1 16072.552,E2 16072.552} C_VEL
LIN {X 0,Y 354.707,Z 1120.128,A -85,B 0,C 180,E1 16069.372,E2 16069.372} C_VEL
LIN {X 0,Y 362.987,Z 1103.575,A -85,B 0,C 180,E1 16065.742,E2 16065.742} C_VEL
LIN {X 0,Y 371.223,Z 1086.895,A -85,B 0,C 180,E1 16062.667,E2 16062.667} C_VEL
LIN {X 0,Y 378.624,Z 1071.81,A -85,B 0,C 180,E1 16060.255,E2 16060.255} C_VEL
LIN {X 0,Y 386.617,Z 1055.144,A -85,B 0,C 180,E1 16057.928,E2 16057.928} C_VEL
LIN {X 0,Y 396.506,Z 1033.627,A -85,B 0,C 180,E1 16055.359,E2 16055.359} C_VEL
LIN {X 0,Y 405.139,Z 1013.552,A -85,B 0,C 180,E1 16053.343,E2 16053.343} C_VEL
LIN {X 0,Y 412.779,Z 994.736,A -85,B 0,C 180,E1 16051.712,E2 16051.712} C_VEL
LIN {X 0,Y 420.399,Z 974.646,A -85,B 0,C 180,E1 16050.208,E2 16050.208} C_VEL
LIN {X 0,Y 429.242,Z 948.758,A -85,B 0,C 180,E1 16048.578,E2 16048.578} C_VEL
LIN {X 0,Y 435.727,Z 927.461,A -85,B 0,C 180,E1 16047.468,E2 16047.468} C_VEL
LIN {X 0,Y 441.219,Z 907.336,A -85,B 0,C 180,E1 16046.578,E2 16046.578} C_VEL
LIN {X 0,Y 446.389,Z 885.912,A -85,B 0,C 180,E1 16045.785,E2 16045.785} C_VEL
LIN {X 0,Y 451.868,Z 859.016,A -85,B 0,C 180,E1 16044.985,E2 16044.985} C_VEL
LIN {X 0,Y 455.838,Z 833.405,A -85,B 0,C 180,E1 16044.409,E2 16044.409} C_VEL
LIN {X 0,Y 458.276,Z 810.916,A -85,B 0,C 180,E1 16043.985,E2 16043.985} C_VEL
LIN {X 0,Y 473.622,Z 596.777,A -85,B 0,C 180,E1 16040.577,E2 16040.577} C_VEL
LIN {X 0,Y 479.283,Z 519.139,A -85,B 0,C 180,E1 16039.341,E2 16039.341} C_VEL
LIN {X 0,Y 470.707,Z 504.048,A -85,B 0,C 180,E1 16036.506,E2 16036.506} C_VEL
LIN {X 0,Y 463.289,Z 491.697,A -85,B 0,C 180,E1 16033.702,E2 16033.702} C_VEL
LIN {X 0,Y 456.56,Z 480.859,A -85,B 0,C 180,E1 16030.729,E2 16030.729} C_VEL
LIN {X 0,Y 451.901,Z 473.963,A -85,B 0,C 180,E1 16028.333,E2 16028.333} C_VEL
LIN {X 0,Y 449.28,Z 469.906,A -85,B 0,C 180,E1 16026.774,E2 16026.774} C_VEL
LIN {X 0,Y 446.487,Z 465.781,A -85,B 0,C 180,E1 16024.882,E2 16024.882} C_VEL
LIN {X 0,Y 443.943,Z 462.007,A -85,B 0,C 180,E1 16022.84,E2 16022.84} C_VEL
LIN {X 0,Y 440.825,Z 457.253,A -85,B 0,C 180,E1 16019.48,E2 16019.48} C_VEL
LIN {X 0,Y 438.415,Z 454.247,A -85,B 0,C 180,E1 16014.241,E2 16014.241} C_VEL
LIN {X 0,Y 438.429,Z 454.276,A -85,B 0,C 180,E1 16011.343,E2 16011.343} C_VEL
LIN {X 0,Y 441.085,Z 457.436,A -85,B 0,C 180,E1 16005.828,E2 16005.828} C_VEL
LIN {X 0,Y 444.862,Z 463.259,A -85,B 0,C 180,E1 16001.998,E2 16001.998} C_VEL
LIN {X 0,Y 448.775,Z 469.058,A -85,B 0,C 180,E1 15999.184,E2 15999.184} C_VEL
LIN {X 0,Y 451.698,Z 473.52,A -85,B 0,C 180,E1 15997.414,E2 15997.414} C_VEL
LIN {X 0,Y 456.446,Z 480.669,A -85,B 0,C 180,E1 15994.955,E2 15994.955} C_VEL
LIN {X 0,Y 462.337,Z 490.208,A -85,B 0,C 180,E1 15992.326,E2 15992.326} C_VEL
LIN {X 0,Y 469.056,Z 501.46,A -85,B 0,C 180,E1 15989.725,E2 15989.725} C_VEL
LIN {X 0,Y 475.513,Z 512.816,A -85,B 0,C 180,E1 15987.503,E2 15987.503} C_VEL
LIN {X 0,Y 475.758,Z 513.709,A -85,B 0,C 180,E1 15987.407,E2 15987.407} C_VEL
LIN {X 0,Y 458.475,Z 748.024,A -85,B 0,C 180,E1 15983.769,E2 15983.769} C_VEL
LIN {X 0,Y 454.57,Z 798.263,A -85,B 0,C 180,E1 15982.96,E2 15982.96} C_VEL
LIN {X 0,Y 450.967,Z 825.656,A -85,B 0,C 180,E1 15982.367,E2 15982.367} C_VEL
LIN {X 0,Y 447.299,Z 846.964,A -85,B 0,C 180,E1 15981.757,E2 15981.757} C_VEL
LIN {X 0,Y 442.98,Z 867.614,A -85,B 0,C 180,E1 15981.039,E2 15981.039} C_VEL
LIN {X 0,Y 436.665,Z 893.066,A -85,B 0,C 180,E1 15979.951,E2 15979.951} C_VEL
LIN {X 0,Y 430.068,Z 915.45,A -85,B 0,C 180,E1 15978.772,E2 15978.772} C_VEL
LIN {X 0,Y 423.819,Z 934.412,A -85,B 0,C 180,E1 15977.597,E2 15977.597} C_VEL
LIN {X 0,Y 415.745,Z 956.658,A -85,B 0,C 180,E1 15975.979,E2 15975.979} C_VEL
LIN {X 0,Y 407.095,Z 977.764,A -85,B 0,C 180,E1 15974.131,E2 15974.131} C_VEL
LIN {X 0,Y 399.632,Z 994.751,A -85,B 0,C 180,E1 15972.398,E2 15972.398} C_VEL
LIN {X 0,Y 391.504,Z 1012.154,A -85,B 0,C 180,E1 15970.346,E2 15970.346} C_VEL
LIN {X 0,Y 381.714,Z 1031.706,A -85,B 0,C 180,E1 15967.612,E2 15967.612} C_VEL
LIN {X 0,Y 374.195,Z 1046.038,A -85,B 0,C 180,E1 15965.251,E2 15965.251} C_VEL
LIN {X 0,Y 366.853,Z 1059.665,A -85,B 0,C 180,E1 15962.66,E2 15962.66} C_VEL
LIN {X 0,Y 358.431,Z 1075.039,A -85,B 0,C 180,E1 15959.22,E2 15959.22} C_VEL
LIN {X 0,Y 351.376,Z 1087.701,A -85,B 0,C 180,E1 15955.809,E2 15955.809} C_VEL
LIN {X 0,Y 345.847,Z 1097.837,A -85,B 0,C 180,E1 15952.613,E2 15952.613} C_VEL
LIN {X 0,Y 340.168,Z 1108.798,A -85,B 0,C 180,E1 15948.508,E2 15948.508} C_VEL
LIN {X 0,Y 335.891,Z 1117.478,A -85,B 0,C 180,E1 15944.48,E2 15944.48} C_VEL
LIN {X 0,Y 333.098,Z 1123.88,A -85,B 0,C 180,E1 15940.901,E2 15940.901} C_VEL
LIN {X 0,Y 330.802,Z 1130.138,A -85,B 0,C 180,E1 15936.595,E2 15936.595} C_VEL
LIN {X 0,Y 329.413,Z 1134.748,A -85,B 0,C 180,E1 15932.261,E2 15932.261} C_VEL
LIN {X 0,Y 328.839,Z 1137.547,A -85,B 0,C 180,E1 15928.606,E2 15928.606} C_VEL
LIN {X 0,Y 328.579,Z 1139.312,A -85,B 0,C 180,E1 15925.112,E2 15925.112} C_VEL
LIN {X 0,Y 328.529,Z 1140.196,A -85,B 0,C 180,E1 15921.6,E2 15921.6} C_VEL
LIN {X 0,Y 328.59,Z 1140.2,A -85,B 0,C 180,E1 15918.058,E2 15918.058} C_VEL
LIN {X 0,Y 328.893,Z 1139.114,A -85,B 0,C 180,E1 15913.883,E2 15913.883} C_VEL
LIN {X 0,Y 329.692,Z 1136.444,A -85,B 0,C 180,E1 15909.403,E2 15909.403} C_VEL
LIN {X 0,Y 331.026,Z 1133.008,A -85,B 0,C 180,E1 15905.556,E2 15905.556} C_VEL
LIN {X 0,Y 333.039,Z 1128.685,A -85,B 0,C 180,E1 15901.878,E2 15901.878} C_VEL
LIN {X 0,Y 336.61,Z 1122.128,A -85,B 0,C 180,E1 15897.477,E2 15897.477} C_VEL
LIN {X 0,Y 341.7,Z 1113.471,A -85,B 0,C 180,E1 15893.022,E2 15893.022} C_VEL
LIN {X 0,Y 346.995,Z 1105.104,A -85,B 0,C 180,E1 15889.473,E2 15889.473} C_VEL
LIN {X 0,Y 348.03,Z 1102.417,A -85,B 0,C 180,E1 15888.286,E2 15888.286} C_VEL
LIN {X 0,Y 348.071,Z 1095.334,A -85,B 0,C 180,E1 15884.986,E2 15884.986} C_VEL
LIN {X 0,Y 349.384,Z 1092.541,A -85,B 0,C 180,E1 15884.016,E2 15884.016} C_VEL
LIN {X 0,Y 356.974,Z 1081.543,A -85,B 0,C 180,E1 15880.865,E2 15880.865} C_VEL
LIN {X 0,Y 365.171,Z 1069.587,A -85,B 0,C 180,E1 15877.949,E2 15877.949} C_VEL
LIN {X 0,Y 375.792,Z 1053.729,A -85,B 0,C 180,E1 15874.7,E2 15874.7} C_VEL
LIN {X 0,Y 385.715,Z 1038.056,A -85,B 0,C 180,E1 15872.042,E2 15872.042} C_VEL
LIN {X 0,Y 394.559,Z 1023.475,A -85,B 0,C 180,E1 15869.926,E2 15869.926} C_VEL
LIN {X 0,Y 404.865,Z 1005.569,A -85,B 0,C 180,E1 15867.705,E2 15867.705} C_VEL
LIN {X 0,Y 415.7,Z 984.997,A -85,B 0,C 180,E1 15865.583,E2 15865.583} C_VEL
LIN {X 0,Y 424.247,Z 967.383,A -85,B 0,C 180,E1 15864.041,E2 15864.041} C_VEL
LIN {X 0,Y 432.722,Z 948.402,A -85,B 0,C 180,E1 15862.617,E2 15862.617} C_VEL
LIN {X 0,Y 442.723,Z 923.244,A -85,B 0,C 180,E1 15861.045,E2 15861.045} C_VEL
LIN {X 0,Y 449.997,Z 902.309,A -85,B 0,C 180,E1 15859.97,E2 15859.97} C_VEL
LIN {X 0,Y 455.877,Z 883.135,A -85,B 0,C 180,E1 15859.135,E2 15859.135} C_VEL
LIN {X 0,Y 462.221,Z 859.189,A -85,B 0,C 180,E1 15858.263,E2 15858.263} C_VEL
LIN {X 0,Y 467.528,Z 833.728,A -85,B 0,C 180,E1 15857.535,E2 15857.535} C_VEL
LIN {X 0,Y 471.177,Z 811.687,A -85,B 0,C 180,E1 15857.048,E2 15857.048} C_VEL
LIN {X 0,Y 474.193,Z 786.497,A -85,B 0,C 180,E1 15856.611,E2 15856.611} C_VEL
LIN {X 0,Y 495.273,Z 547.721,A -85,B 0,C 180,E1 15853.008,E2 15853.008} C_VEL
LIN {X 0,Y 496.549,Z 533.67,A -85,B 0,C 180,E1 15852.797,E2 15852.797} C_VEL
LIN {X 0,Y 492.288,Z 526.057,A -85,B 0,C 180,E1 15850.415,E2 15850.415} C_VEL
LIN {X 0,Y 488.994,Z 520.142,A -85,B 0,C 180,E1 15848.17,E2 15848.17} C_VEL
LIN {X 0,Y 486.56,Z 516.066,A -85,B 0,C 180,E1 15846.134,E2 15846.134} C_VEL
LIN {X 0,Y 484.187,Z 511.955,A -85,B 0,C 180,E1 15843.433,E2 15843.433} C_VEL
LIN {X 0,Y 482.247,Z 508.716,A -85,B 0,C 180,E1 15838.693,E2 15838.693} C_VEL
LIN {X 0,Y 482.313,Z 508.958,A -85,B 0,C 180,E1 15836.434,E2 15836.434} C_VEL
LIN {X 0,Y 484.622,Z 512.746,A -85,B 0,C 180,E1 15831.636,E2 15831.636} C_VEL
LIN {X 0,Y 487.528,Z 517.85,A -85,B 0,C 180,E1 15828.645,E2 15828.645} C_VEL
LIN {X 0,Y 491.216,Z 524.2,A -85,B 0,C 180,E1 15825.922,E2 15825.922} C_VEL
LIN {X 0,Y 496.119,Z 533.086,A -85,B 0,C 180,E1 15823.068,E2 15823.068} C_VEL
LIN {X 0,Y 497.585,Z 536.036,A -85,B 0,C 180,E1 15822.31,E2 15822.31} C_VEL
LIN {X 0,Y 478.387,Z 754.301,A -85,B 0,C 180,E1 15818.92,E2 15818.92} C_VEL
LIN {X 0,Y 472.914,Z 815.328,A -85,B 0,C 180,E1 15817.947,E2 15817.947} C_VEL
LIN {X 0,Y 468.535,Z 844.761,A -85,B 0,C 180,E1 15817.382,E2 15817.382} C_VEL
LIN {X 0,Y 463.936,Z 867.325,A -85,B 0,C 180,E1 15816.855,E2 15816.855} C_VEL
LIN {X 0,Y 458.825,Z 888.33,A -85,B 0,C 180,E1 15816.241,E2 15816.241} C_VEL
LIN {X 0,Y 452.036,Z 912.334,A -85,B 0,C 180,E1 15815.38,E2 15815.38} C_VEL
LIN {X 0,Y 443.499,Z 937.957,A -85,B 0,C 180,E1 15814.231,E2 15814.231} C_VEL
LIN {X 0,Y 435.935,Z 958.161,A -85,B 0,C 180,E1 15813.137,E2 15813.137} C_VEL
LIN {X 0,Y 428.011,Z 977.519,A -85,B 0,C 180,E1 15811.907,E2 15811.907} C_VEL
LIN {X 0,Y 418.408,Z 999.102,A -85,B 0,C 180,E1 15810.302,E2 15810.302} C_VEL
LIN {X 0,Y 407.028,Z 1022.418,A -85,B 0,C 180,E1 15808.206,E2 15808.206} C_VEL
LIN {X 0,Y 397.747,Z 1040.217,A -85,B 0,C 180,E1 15806.312,E2 15806.312} C_VEL
LIN {X 0,Y 388.373,Z 1057.403,A -85,B 0,C 180,E1 15804.19,E2 15804.19} C_VEL
LIN {X 0,Y 377.444,Z 1076.739,A -85,B 0,C 180,E1 15801.395,E2 15801.395} C_VEL
LIN {X 0,Y 366.932,Z 1094.514,A -85,B 0,C 180,E1 15798.299,E2 15798.299} C_VEL
LIN {X 0,Y 358.786,Z 1108.242,A -85,B 0,C 180,E1 15795.514,E2 15795.514} C_VEL
LIN {X 0,Y 350.677,Z 1121.986,A -85,B 0,C 180,E1 15792.291,E2 15792.291} C_VEL
LIN {X 0,Y 341.633,Z 1137.682,A -85,B 0,C 180,E1 15787.924,E2 15787.924} C_VEL
LIN {X 0,Y 335.372,Z 1149.172,A -85,B 0,C 180,E1 15784.09,E2 15784.09} C_VEL
LIN {X 0,Y 330.504,Z 1158.806,A -85,B 0,C 180,E1 15780.346,E2 15780.346} C_VEL
LIN {X 0,Y 326.583,Z 1167.579,A -85,B 0,C 180,E1 15776.355,E2 15776.355} C_VEL
LIN {X 0,Y 323.145,Z 1176.83,A -85,B 0,C 180,E1 15771.224,E2 15771.224} C_VEL
LIN {X 0,Y 321.44,Z 1182.852,A -85,B 0,C 180,E1 15767.001,E2 15767.001} C_VEL
LIN {X 0,Y 320.65,Z 1187.026,A -85,B 0,C 180,E1 15763.341,E2 15763.341} C_VEL
LIN {X 0,Y 320.337,Z 1190.194,A -85,B 0,C 180,E1 15759.704,E2 15759.704} C_VEL
LIN {X 0,Y 320.291,Z 1192.278,A -85,B 0,C 180,E1 15756.273,E2 15756.273} C_VEL
LIN {X 0,Y 320.344,Z 1193.464,A -85,B 0,C 180,E1 15752.781,E2 15752.781} C_VEL
LIN {X 0,Y 320.36,Z 1193.68,A -85,B 0,C 180,E1 15749.285,E2 15749.285} C_VEL
LIN {X 0,Y 320.329,Z 1192.948,A -85,B 0,C 180,E1 15745.883,E2 15745.883} C_VEL
LIN {X 0,Y 320.317,Z 1191.155,A -85,B 0,C 180,E1 15742.286,E2 15742.286} C_VEL
LIN {X 0,Y 320.453,Z 1188.317,A -85,B 0,C 180,E1 15738.664,E2 15738.664} C_VEL
LIN {X 0,Y 320.999,Z 1184.325,A -85,B 0,C 180,E1 15734.935,E2 15734.935} C_VEL
LIN {X 0,Y 322.073,Z 1179.173,A -85,B 0,C 180,E1 15731.164,E2 15731.164} C_VEL
LIN {X 0,Y 323.831,Z 1173.047,A -85,B 0,C 180,E1 15727.489,E2 15727.489} C_VEL
LIN {X 0,Y 326.667,Z 1165.009,A -85,B 0,C 180,E1 15723.457,E2 15723.457} C_VEL
LIN {X 0,Y 331.621,Z 1153.093,A -85,B 0,C 180,E1 15718.56,E2 15718.56} C_VEL
LIN {X 0,Y 336.387,Z 1142.716,A -85,B 0,C 180,E1 15714.994,E2 15714.994} C_VEL
LIN {X 0,Y 341.863,Z 1131.569,A -85,B 0,C 180,E1 15711.681,E2 15711.681} C_VEL
LIN {X 0,Y 348.595,Z 1118.381,A -85,B 0,C 180,E1 15708.285,E2 15708.285} C_VEL
LIN {X 0,Y 357.542,Z 1101.056,A -85,B 0,C 180,E1 15704.512,E2 15704.512} C_VEL
LIN {X 0,Y 365.464,Z 1085.638,A -85,B 0,C 180,E1 15701.67,E2 15701.67} C_VEL
LIN {X 0,Y 373.228,Z 1070.33,A -85,B 0,C 180,E1 15699.217,E2 15699.217} C_VEL
LIN {X 0,Y 382.475,Z 1051.63,A -85,B 0,C 180,E1 15696.626,E2 15696.626} C_VEL
LIN {X 0,Y 392.526,Z 1030.068,A -85,B 0,C 180,E1 15694.122,E2 15694.122} C_VEL
LIN {X 0,Y 400.722,Z 1011.446,A -85,B 0,C 180,E1 15692.275,E2 15692.275} C_VEL
LIN {X 0,Y 408.543,Z 992.56,A -85,B 0,C 180,E1 15690.655,E2 15690.655} C_VEL
LIN {X 0,Y 417.907,Z 968.104,A -85,B 0,C 180,E1 15688.876,E2 15688.876} C_VEL
LIN {X 0,Y 425.704,Z 945.207,A -85,B 0,C 180,E1 15687.499,E2 15687.499} C_VEL
LIN {X 0,Y 431.853,Z 925.255,A -85,B 0,C 180,E1 15686.48,E2 15686.48} C_VEL
LIN {X 0,Y 437.775,Z 903.8,A -85,B 0,C 180,E1 15685.557,E2 15685.557} C_VEL
LIN {X 0,Y 444.256,Z 876.356,A -85,B 0,C 180,E1 15684.597,E2 15684.597} C_VEL
LIN {X 0,Y 448.887,Z 852.11,A -85,B 0,C 180,E1 15683.945,E2 15683.945} C_VEL
LIN {X 0,Y 452.242,Z 829.884,A -85,B 0,C 180,E1 15683.464,E2 15683.464} C_VEL
LIN {X 0,Y 454.904,Z 804.066,A -85,B 0,C 180,E1 15682.992,E2 15682.992} C_VEL
LIN {X 0,Y 471.329,Z 579.536,A -85,B 0,C 180,E1 15679.433,E2 15679.433} C_VEL
LIN {X 0,Y 475.516,Z 523.724,A -85,B 0,C 180,E1 15678.545,E2 15678.545} C_VEL
LIN {X 0,Y 467.541,Z 509.476,A -85,B 0,C 180,E1 15675.792,E2 15675.792} C_VEL
LIN {X 0,Y 460.233,Z 497.143,A -85,B 0,C 180,E1 15672.899,E2 15672.899} C_VEL
LIN {X 0,Y 454.392,Z 487.655,A -85,B 0,C 180,E1 15670.203,E2 15670.203} C_VEL
LIN {X 0,Y 448.676,Z 478.658,A -85,B 0,C 180,E1 15667.04,E2 15667.04} C_VEL
LIN {X 0,Y 445.048,Z 473.318,A -85,B 0,C 180,E1 15664.575,E2 15664.575} C_VEL
LIN {X 0,Y 442.797,Z 469.87,A -85,B 0,C 180,E1 15662.718,E2 15662.718} C_VEL
LIN {X 0,Y 439.735,Z 465.126,A -85,B 0,C 180,E1 15659.349,E2 15659.349} C_VEL
LIN {X 0,Y 437.417,Z 462.151,A -85,B 0,C 180,E1 15654.096,E2 15654.096} C_VEL
LIN {X 0,Y 437.473,Z 462.276,A -85,B 0,C 180,E1 15651.191,E2 15651.191} C_VEL
LIN {X 0,Y 440.01,Z 465.369,A -85,B 0,C 180,E1 15645.927,E2 15645.927} C_VEL
LIN {X 0,Y 443.588,Z 470.978,A -85,B 0,C 180,E1 15642.216,E2 15642.216} C_VEL
LIN {X 0,Y 447.52,Z 476.923,A -85,B 0,C 180,E1 15639.328,E2 15639.328} C_VEL
LIN {X 0,Y 451.77,Z 483.398,A -85,B 0,C 180,E1 15636.799,E2 15636.799} C_VEL
LIN {X 0,Y 457.628,Z 492.79,A -85,B 0,C 180,E1 15633.894,E2 15633.894} C_VEL
LIN {X 0,Y 464.442,Z 504.278,A -85,B 0,C 180,E1 15631.027,E2 15631.027} C_VEL
LIN {X 0,Y 471.409,Z 516.569,A -85,B 0,C 180,E1 15628.477,E2 15628.477} C_VEL
LIN {X 0,Y 472.124,Z 518.083,A -85,B 0,C 180,E1 15628.224,E2 15628.224} C_VEL
LIN {X 0,Y 454.42,Z 752.207,A -85,B 0,C 180,E1 15624.594,E2 15624.594} C_VEL
LIN {X 0,Y 450.608,Z 799.623,A -85,B 0,C 180,E1 15623.829,E2 15623.829} C_VEL
LIN {X 0,Y 446.959,Z 826.414,A -85,B 0,C 180,E1 15623.245,E2 15623.245} C_VEL
LIN {X 0,Y 443.247,Z 847.497,A -85,B 0,C 180,E1 15622.643,E2 15622.643} C_VEL
LIN {X 0,Y 438.823,Z 868.189,A -85,B 0,C 180,E1 15621.926,E2 15621.926} C_VEL
LIN {X 0,Y 432.172,Z 894.284,A -85,B 0,C 180,E1 15620.809,E2 15620.809} C_VEL
LIN {X 0,Y 425.626,Z 915.99,A -85,B 0,C 180,E1 15619.667,E2 15619.667} C_VEL
LIN {X 0,Y 419.235,Z 934.961,A -85,B 0,C 180,E1 15618.493,E2 15618.493} C_VEL
LIN {X 0,Y 410.966,Z 957.218,A -85,B 0,C 180,E1 15616.876,E2 15616.876} C_VEL
LIN {X 0,Y 402.097,Z 978.321,A -85,B 0,C 180,E1 15615.027,E2 15615.027} C_VEL
LIN {X 0,Y 394.431,Z 995.31,A -85,B 0,C 180,E1 15613.29,E2 15613.29} C_VEL
LIN {X 0,Y 386.071,Z 1012.72,A -85,B 0,C 180,E1 15611.232,E2 15611.232} C_VEL
LIN {X 0,Y 375.991,Z 1032.288,A -85,B 0,C 180,E1 15608.482,E2 15608.482} C_VEL
LIN {X 0,Y 368.228,Z 1046.623,A -85,B 0,C 180,E1 15606.102,E2 15606.102} C_VEL
LIN {X 0,Y 360.63,Z 1060.253,A -85,B 0,C 180,E1 15603.486,E2 15603.486} C_VEL
LIN {X 0,Y 351.891,Z 1075.64,A -85,B 0,C 180,E1 15600.005,E2 15600.005} C_VEL
LIN {X 0,Y 344.87,Z 1087.772,A -85,B 0,C 180,E1 15596.704,E2 15596.704} C_VEL
LIN {X 0,Y 339.064,Z 1097.966,A -85,B 0,C 180,E1 15593.459,E2 15593.459} C_VEL
LIN {X 0,Y 333.064,Z 1109.038,A -85,B 0,C 180,E1 15589.282,E2 15589.282} C_VEL
LIN {X 0,Y 328.356,Z 1118.105,A -85,B 0,C 180,E1 15585,E2 15585} C_VEL
LIN {X 0,Y 325.29,Z 1124.791,A -85,B 0,C 180,E1 15581.166,E2 15581.166} C_VEL
LIN {X 0,Y 322.824,Z 1131.201,A -85,B 0,C 180,E1 15576.58,E2 15576.58} C_VEL
LIN {X 0,Y 321.457,Z 1135.534,A -85,B 0,C 180,E1 15572.317,E2 15572.317} C_VEL
LIN {X 0,Y 320.865,Z 1138.296,A -85,B 0,C 180,E1 15568.571,E2 15568.571} C_VEL
LIN {X 0,Y 320.602,Z 1140.025,A -85,B 0,C 180,E1 15564.99,E2 15564.99} C_VEL
LIN {X 0,Y 320.553,Z 1140.877,A -85,B 0,C 180,E1 15561.389,E2 15561.389} C_VEL
LIN {X 0,Y 320.654,Z 1140.818,A -85,B 0,C 180,E1 15557.392,E2 15557.392} C_VEL
LIN {X 0,Y 321.063,Z 1139.386,A -85,B 0,C 180,E1 15552.791,E2 15552.791} C_VEL
LIN {X 0,Y 321.931,Z 1136.851,A -85,B 0,C 180,E1 15548.692,E2 15548.692} C_VEL
LIN {X 0,Y 323.355,Z 1133.53,A -85,B 0,C 180,E1 15544.936,E2 15544.936} C_VEL
LIN {X 0,Y 325.688,Z 1128.935,A -85,B 0,C 180,E1 15540.984,E2 15540.984} C_VEL
LIN {X 0,Y 329.99,Z 1121.562,A -85,B 0,C 180,E1 15536.116,E2 15536.116} C_VEL
LIN {X 0,Y 334.968,Z 1113.682,A -85,B 0,C 180,E1 15532.055,E2 15532.055} C_VEL
LIN {X 0,Y 340.629,Z 1105.231,A -85,B 0,C 180,E1 15528.441,E2 15528.441} C_VEL
LIN {X 0,Y 348.9,Z 1093.271,A -85,B 0,C 180,E1 15524.239,E2 15524.239} C_VEL
LIN {X 0,Y 349.384,Z 1092.541,A -85,B 0,C 180,E1 15524.016,E2 15524.016} C_VEL
LIN {X 0,Y 350.904,Z 1089.306,A -85,B 0,C 180,E1 15522.893,E2 15522.893} C_VEL
LIN {X 0,Y 352.254,Z 1081.542,A -85,B 0,C 180,E1 15519.874,E2 15519.874} C_VEL
LIN {X 0,Y 354.207,Z 1077.948,A -85,B 0,C 180,E1 15518.799,E2 15518.799} C_VEL
LIN {X 0,Y 364.53,Z 1063.195,A -85,B 0,C 180,E1 15515.449,E2 15515.449} C_VEL
LIN {X 0,Y 373.733,Z 1049.601,A -85,B 0,C 180,E1 15512.854,E2 15512.854} C_VEL
LIN {X 0,Y 383.334,Z 1034.853,A -85,B 0,C 180,E1 15510.452,E2 15510.452} C_VEL
LIN {X 0,Y 395.663,Z 1014.653,A -85,B 0,C 180,E1 15507.71,E2 15507.71} C_VEL
LIN {X 0,Y 405.305,Z 997.616,A -85,B 0,C 180,E1 15505.785,E2 15505.785} C_VEL
LIN {X 0,Y 414.208,Z 980.763,A -85,B 0,C 180,E1 15504.153,E2 15504.153} C_VEL
LIN {X 0,Y 424.504,Z 959.63,A -85,B 0,C 180,E1 15502.41,E2 15502.41} C_VEL
LIN {X 0,Y 433.828,Z 937.946,A -85,B 0,C 180,E1 15500.931,E2 15500.931} C_VEL
LIN {X 0,Y 441.12,Z 919.146,A -85,B 0,C 180,E1 15499.838,E2 15499.838} C_VEL
LIN {X 0,Y 448.766,Z 897.056,A -85,B 0,C 180,E1 15498.754,E2 15498.754} C_VEL
LIN {X 0,Y 456.212,Z 871.583,A -85,B 0,C 180,E1 15497.737,E2 15497.737} C_VEL
LIN {X 0,Y 461.463,Z 850.099,A -85,B 0,C 180,E1 15497.047,E2 15497.047} C_VEL
LIN {X 0,Y 465.568,Z 829.781,A -85,B 0,C 180,E1 15496.509,E2 15496.509} C_VEL
LIN {X 0,Y 469.734,Z 803.531,A -85,B 0,C 180,E1 15495.969,E2 15495.969} C_VEL
LIN {X 0,Y 474.035,Z 758.795,A -85,B 0,C 180,E1 15495.27,E2 15495.27} C_VEL
LIN {X 0,Y 493.951,Z 539.222,A -85,B 0,C 180,E1 15491.981,E2 15491.981} C_VEL
LIN {X 0,Y 489.52,Z 531.104,A -85,B 0,C 180,E1 15489.286,E2 15489.286} C_VEL
LIN {X 0,Y 485.838,Z 524.466,A -85,B 0,C 180,E1 15486.381,E2 15486.381} C_VEL
LIN {X 0,Y 483.121,Z 519.835,A -85,B 0,C 180,E1 15483.322,E2 15483.322} C_VEL
LIN {X 0,Y 481.258,Z 516.627,A -85,B 0,C 180,E1 15478.571,E2 15478.571} C_VEL
LIN {X 0,Y 481.35,Z 516.98,A -85,B 0,C 180,E1 15476.308,E2 15476.308} C_VEL
LIN {X 0,Y 483.5,Z 520.552,A -85,B 0,C 180,E1 15471.796,E2 15471.796} C_VEL
LIN {X 0,Y 486.265,Z 525.544,A -85,B 0,C 180,E1 15468.855,E2 15468.855} C_VEL
LIN {X 0,Y 489.776,Z 531.761,A -85,B 0,C 180,E1 15466.181,E2 15466.181} C_VEL
LIN {X 0,Y 494.511,Z 540.562,A -85,B 0,C 180,E1 15463.344,E2 15463.344} C_VEL
LIN {X 0,Y 494.903,Z 541.609,A -85,B 0,C 180,E1 15463.118,E2 15463.118} C_VEL
LIN {X 0,Y 475.282,Z 759.769,A -85,B 0,C 180,E1 15459.746,E2 15459.746} C_VEL
LIN {X 0,Y 470.102,Z 815.741,A -85,B 0,C 180,E1 15458.856,E2 15458.856} C_VEL
LIN {X 0,Y 465.701,Z 844.532,A -85,B 0,C 180,E1 15458.307,E2 15458.307} C_VEL
LIN {X 0,Y 461.051,Z 866.954,A -85,B 0,C 180,E1 15457.791,E2 15457.791} C_VEL
LIN {X 0,Y 455.822,Z 888.042,A -85,B 0,C 180,E1 15457.185,E2 15457.185} C_VEL
LIN {X 0,Y 448.742,Z 912.574,A -85,B 0,C 180,E1 15456.314,E2 15456.314} C_VEL
LIN {X 0,Y 440.012,Z 938.078,A -85,B 0,C 180,E1 15455.178,E2 15455.178} C_VEL
LIN {X 0,Y 432.353,Z 958.067,A -85,B 0,C 180,E1 15454.106,E2 15454.106} C_VEL
LIN {X 0,Y 424.469,Z 976.873,A -85,B 0,C 180,E1 15452.923,E2 15452.923} C_VEL
LIN {X 0,Y 414.514,Z 998.714,A -85,B 0,C 180,E1 15451.313,E2 15451.313} C_VEL
LIN {X 0,Y 402.995,Z 1021.687,A -85,B 0,C 180,E1 15449.262,E2 15449.262} C_VEL
LIN {X 0,Y 393.663,Z 1039.117,A -85,B 0,C 180,E1 15447.42,E2 15447.42} C_VEL
LIN {X 0,Y 384.126,Z 1056.083,A -85,B 0,C 180,E1 15445.339,E2 15445.339} C_VEL
LIN {X 0,Y 373.341,Z 1074.55,A -85,B 0,C 180,E1 15442.694,E2 15442.694} C_VEL
LIN {X 0,Y 361.846,Z 1093.331,A -85,B 0,C 180,E1 15439.454,E2 15439.454} C_VEL
LIN {X 0,Y 352.825,Z 1107.923,A -85,B 0,C 180,E1 15436.476,E2 15436.476} C_VEL
LIN {X 0,Y 344.428,Z 1121.536,A -85,B 0,C 180,E1 15433.243,E2 15433.243} C_VEL
LIN {X 0,Y 334.642,Z 1137.729,A -85,B 0,C 180,E1 15428.643,E2 15428.643} C_VEL
LIN {X 0,Y 328.371,Z 1148.647,A -85,B 0,C 180,E1 15424.921,E2 15424.921} C_VEL
LIN {X 0,Y 323.243,Z 1158.265,A -85,B 0,C 180,E1 15421.102,E2 15421.102} C_VEL
LIN {X 0,Y 318.909,Z 1167.394,A -85,B 0,C 180,E1 15416.839,E2 15416.839} C_VEL
LIN {X 0,Y 315.295,Z 1176.515,A -85,B 0,C 180,E1 15411.584,E2 15411.584} C_VEL
LIN {X 0,Y 313.559,Z 1182.244,A -85,B 0,C 180,E1 15407.442,E2 15407.442} C_VEL
LIN {X 0,Y 312.708,Z 1186.407,A -85,B 0,C 180,E1 15403.687,E2 15403.687} C_VEL
LIN {X 0,Y 312.362,Z 1189.565,A -85,B 0,C 180,E1 15399.954,E2 15399.954} C_VEL
LIN {X 0,Y 312.309,Z 1191.639,A -85,B 0,C 180,E1 15396.434,E2 15396.434} C_VEL
LIN {X 0,Y 312.367,Z 1192.806,A -85,B 0,C 180,E1 15392.897,E2 15392.897} C_VEL
LIN {X 0,Y 312.387,Z 1193.035,A -85,B 0,C 180,E1 15389.45,E2 15389.45} C_VEL
LIN {X 0,Y 312.355,Z 1192.335,A -85,B 0,C 180,E1 15385.962,E2 15385.962} C_VEL
LIN {X 0,Y 312.337,Z 1190.571,A -85,B 0,C 180,E1 15382.273,E2 15382.273} C_VEL
LIN {X 0,Y 312.475,Z 1187.757,A -85,B 0,C 180,E1 15378.557,E2 15378.557} C_VEL
LIN {X 0,Y 313.049,Z 1183.759,A -85,B 0,C 180,E1 15374.71,E2 15374.71} C_VEL
LIN {X 0,Y 314.171,Z 1178.659,A -85,B 0,C 180,E1 15370.865,E2 15370.865} C_VEL
LIN {X 0,Y 315.907,Z 1172.884,A -85,B 0,C 180,E1 15367.286,E2 15367.286} C_VEL
LIN {X 0,Y 318.599,Z 1165.498,A -85,B 0,C 180,E1 15363.438,E2 15363.438} C_VEL
LIN {X 0,Y 322.654,Z 1155.982,A -85,B 0,C 180,E1 15359.249,E2 15359.249} C_VEL
LIN {X 0,Y 328.724,Z 1143.171,A -85,B 0,C 180,E1 15354.606,E2 15354.606} C_VEL
LIN {X 0,Y 334.539,Z 1131.787,A -85,B 0,C 180,E1 15351.124,E2 15351.124} C_VEL
LIN {X 0,Y 340.993,Z 1119.584,A -85,B 0,C 180,E1 15347.891,E2 15347.891} C_VEL
LIN {X 0,Y 349.632,Z 1103.605,A -85,B 0,C 180,E1 15344.251,E2 15344.251} C_VEL
LIN {X 0,Y 359.139,Z 1085.679,A -85,B 0,C 180,E1 15340.865,E2 15340.865} C_VEL
LIN {X 0,Y 367.233,Z 1070.228,A -85,B 0,C 180,E1 15338.36,E2 15338.36} C_VEL
LIN {X 0,Y 376.303,Z 1052.432,A -85,B 0,C 180,E1 15335.865,E2 15335.865} C_VEL
LIN {X 0,Y 386.9,Z 1030.495,A -85,B 0,C 180,E1 15333.279,E2 15333.279} C_VEL
LIN {X 0,Y 395.47,Z 1011.551,A -85,B 0,C 180,E1 15331.389,E2 15331.389} C_VEL
LIN {X 0,Y 403.616,Z 992.392,A -85,B 0,C 180,E1 15329.741,E2 15329.741} C_VEL
LIN {X 0,Y 412.897,Z 968.88,A -85,B 0,C 180,E1 15328.021,E2 15328.021} C_VEL
LIN {X 0,Y 421.146,Z 945.231,A -85,B 0,C 180,E1 15326.598,E2 15326.598} C_VEL
LIN {X 0,Y 427.727,Z 924.309,A -85,B 0,C 180,E1 15325.536,E2 15325.536} C_VEL
LIN {X 0,Y 433.988,Z 902.004,A -85,B 0,C 180,E1 15324.589,E2 15324.589} C_VEL
LIN {X 0,Y 440.687,Z 873.674,A -85,B 0,C 180,E1 15323.627,E2 15323.627} C_VEL
LIN {X 0,Y 445.075,Z 850.92,A -85,B 0,C 180,E1 15323.027,E2 15323.027} C_VEL
LIN {X 0,Y 448.496,Z 828.425,A -85,B 0,C 180,E1 15322.546,E2 15322.546} C_VEL
LIN {X 0,Y 451.367,Z 800.05,A -85,B 0,C 180,E1 15322.036,E2 15322.036} C_VEL
LIN {X 0,Y 468.283,Z 574.436,A -85,B 0,C 180,E1 15318.467,E2 15318.467} C_VEL
LIN {X 0,Y 471.835,Z 528.339,A -85,B 0,C 180,E1 15317.736,E2 15317.736} C_VEL
LIN {X 0,Y 464.67,Z 515.335,A -85,B 0,C 180,E1 15315.156,E2 15315.156} C_VEL
LIN {X 0,Y 457.464,Z 502.919,A -85,B 0,C 180,E1 15312.176,E2 15312.176} C_VEL
LIN {X 0,Y 451.783,Z 493.704,A -85,B 0,C 180,E1 15309.426,E2 15309.426} C_VEL
LIN {X 0,Y 446.849,Z 485.771,A -85,B 0,C 180,E1 15306.553,E2 15306.553} C_VEL
LIN {X 0,Y 443.705,Z 480.975,A -85,B 0,C 180,E1 15304.33,E2 15304.33} C_VEL
LIN {X 0,Y 441.506,Z 477.567,A -85,B 0,C 180,E1 15302.466,E2 15302.466} C_VEL
LIN {X 0,Y 438.647,Z 473,A -85,B 0,C 180,E1 15299.216,E2 15299.216} C_VEL
LIN {X 0,Y 436.437,Z 470.092,A -85,B 0,C 180,E1 15294.082,E2 15294.082} C_VEL
LIN {X 0,Y 436.497,Z 470.233,A -85,B 0,C 180,E1 15291.171,E2 15291.171} C_VEL
LIN {X 0,Y 438.944,Z 473.319,A -85,B 0,C 180,E1 15286.018,E2 15286.018} C_VEL
LIN {X 0,Y 442.393,Z 478.835,A -85,B 0,C 180,E1 15282.37,E2 15282.37} C_VEL
LIN {X 0,Y 446.26,Z 484.774,A -85,B 0,C 180,E1 15279.478,E2 15279.478} C_VEL
LIN {X 0,Y 450.568,Z 491.604,A -85,B 0,C 180,E1 15276.871,E2 15276.871} C_VEL
LIN {X 0,Y 455.815,Z 500.137,A -85,B 0,C 180,E1 15274.222,E2 15274.222} C_VEL
LIN {X 0,Y 462.443,Z 511.561,A -85,B 0,C 180,E1 15271.362,E2 15271.362} C_VEL
LIN {X 0,Y 468.561,Z 522.574,A -85,B 0,C 180,E1 15269.054,E2 15269.054} C_VEL
LIN {X 0,Y 450.801,Z 751.782,A -85,B 0,C 180,E1 15265.505,E2 15265.505} C_VEL
LIN {X 0,Y 446.854,Z 799.789,A -85,B 0,C 180,E1 15264.732,E2 15264.732} C_VEL
LIN {X 0,Y 443.121,Z 826.753,A -85,B 0,C 180,E1 15264.149,E2 15264.149} C_VEL
LIN {X 0,Y 439.34,Z 847.814,A -85,B 0,C 180,E1 15263.551,E2 15263.551} C_VEL
LIN {X 0,Y 434.772,Z 868.756,A -85,B 0,C 180,E1 15262.831,E2 15262.831} C_VEL
LIN {X 0,Y 427.978,Z 894.831,A -85,B 0,C 180,E1 15261.718,E2 15261.718} C_VEL
LIN {X 0,Y 421.29,Z 916.531,A -85,B 0,C 180,E1 15260.58,E2 15260.58} C_VEL
LIN {X 0,Y 414.442,Z 936.367,A -85,B 0,C 180,E1 15259.352,E2 15259.352} C_VEL
LIN {X 0,Y 405.682,Z 959.17,A -85,B 0,C 180,E1 15257.679,E2 15257.679} C_VEL
LIN {X 0,Y 396.909,Z 979.507,A -85,B 0,C 180,E1 15255.885,E2 15255.885} C_VEL
LIN {X 0,Y 389.053,Z 996.448,A -85,B 0,C 180,E1 15254.144,E2 15254.144} C_VEL
LIN {X 0,Y 379.438,Z 1015.909,A -85,B 0,C 180,E1 15251.811,E2 15251.811} C_VEL
LIN {X 0,Y 369.863,Z 1033.729,A -85,B 0,C 180,E1 15249.24,E2 15249.24} C_VEL
LIN {X 0,Y 361.887,Z 1048.001,A -85,B 0,C 180,E1 15246.837,E2 15246.837} C_VEL
LIN {X 0,Y 353.656,Z 1062.295,A -85,B 0,C 180,E1 15244.041,E2 15244.041} C_VEL
LIN {X 0,Y 344.318,Z 1078.022,A -85,B 0,C 180,E1 15240.349,E2 15240.349} C_VEL
LIN {X 0,Y 337.479,Z 1089.448,A -85,B 0,C 180,E1 15237.146,E2 15237.146} C_VEL
LIN {X 0,Y 331.24,Z 1100.023,A -85,B 0,C 180,E1 15233.67,E2 15233.67} C_VEL
LIN {X 0,Y 324.682,Z 1111.541,A -85,B 0,C 180,E1 15229.052,E2 15229.052} C_VEL
LIN {X 0,Y 320.509,Z 1119.381,A -85,B 0,C 180,E1 15225.191,E2 15225.191} C_VEL
LIN {X 0,Y 317.247,Z 1126.263,A -85,B 0,C 180,E1 15221.084,E2 15221.084} C_VEL
LIN {X 0,Y 314.692,Z 1132.6,A -85,B 0,C 180,E1 15216.201,E2 15216.201} C_VEL
LIN {X 0,Y 313.459,Z 1136.468,A -85,B 0,C 180,E1 15212.194,E2 15212.194} C_VEL
LIN {X 0,Y 312.891,Z 1139.044,A -85,B 0,C 180,E1 15208.535,E2 15208.535} C_VEL
LIN {X 0,Y 312.625,Z 1140.738,A -85,B 0,C 180,E1 15204.862,E2 15204.862} C_VEL
LIN {X 0,Y 312.579,Z 1141.558,A -85,B 0,C 180,E1 15201.168,E2 15201.168} C_VEL
LIN {X 0,Y 312.707,Z 1141.456,A -85,B 0,C 180,E1 15196.878,E2 15196.878} C_VEL
LIN {X 0,Y 313.196,Z 1139.869,A -85,B 0,C 180,E1 15192.153,E2 15192.153} C_VEL
LIN {X 0,Y 314.133,Z 1137.407,A -85,B 0,C 180,E1 15188.136,E2 15188.136} C_VEL
LIN {X 0,Y 315.711,Z 1134.054,A -85,B 0,C 180,E1 15184.286,E2 15184.286} C_VEL
LIN {X 0,Y 318.414,Z 1129.188,A -85,B 0,C 180,E1 15180.048,E2 15180.048} C_VEL
LIN {X 0,Y 323.108,Z 1121.642,A -85,B 0,C 180,E1 15175.076,E2 15175.076} C_VEL
LIN {X 0,Y 327.951,Z 1114.444,A -85,B 0,C 180,E1 15171.309,E2 15171.309} C_VEL
LIN {X 0,Y 333.894,Z 1106.025,A -85,B 0,C 180,E1 15167.641,E2 15167.641} C_VEL
LIN {X 0,Y 342.535,Z 1094.105,A -85,B 0,C 180,E1 15163.379,E2 15163.379} C_VEL
LIN {X 0,Y 350.944,Z 1082.399,A -85,B 0,C 180,E1 15159.969,E2 15159.969} C_VEL
LIN {X 0,Y 354.207,Z 1077.948,A -85,B 0,C 180,E1 15158.799,E2 15158.799} C_VEL
LIN {X 0,Y 356.243,Z 1074.302,A -85,B 0,C 180,E1 15157.742,E2 15157.742} C_VEL
LIN {X 0,Y 358.811,Z 1065.343,A -85,B 0,C 180,E1 15154.884,E2 15154.884} C_VEL
LIN {X 0,Y 361.118,Z 1061.219,A -85,B 0,C 180,E1 15153.903,E2 15153.903} C_VEL
LIN {X 0,Y 371.733,Z 1046.013,A -85,B 0,C 180,E1 15151.094,E2 15151.094} C_VEL
LIN {X 0,Y 383.683,Z 1027.731,A -85,B 0,C 180,E1 15148.314,E2 15148.314} C_VEL
LIN {X 0,Y 393.224,Z 1012.182,A -85,B 0,C 180,E1 15146.323,E2 15146.323} C_VEL
LIN {X 0,Y 403.083,Z 995.051,A -85,B 0,C 180,E1 15144.446,E2 15144.446} C_VEL
LIN {X 0,Y 415.143,Z 972.115,A -85,B 0,C 180,E1 15142.354,E2 15142.354} C_VEL
LIN {X 0,Y 423.951,Z 953.54,A -85,B 0,C 180,E1 15140.943,E2 15140.943} C_VEL
LIN {X 0,Y 432.237,Z 934.345,A -85,B 0,C 180,E1 15139.699,E2 15139.699} C_VEL
LIN {X 0,Y 441.104,Z 911.43,A -85,B 0,C 180,E1 15138.446,E2 15138.446} C_VEL
LIN {X 0,Y 448.735,Z 888.147,A -85,B 0,C 180,E1 15137.405,E2 15137.405} C_VEL
LIN {X 0,Y 454.484,Z 867.871,A -85,B 0,C 180,E1 15136.646,E2 15136.646} C_VEL
LIN {X 0,Y 460.011,Z 844.914,A -85,B 0,C 180,E1 15135.945,E2 15135.945} C_VEL
LIN {X 0,Y 465.166,Z 817.253,A -85,B 0,C 180,E1 15135.297,E2 15135.297} C_VEL
LIN {X 0,Y 468.167,Z 794.907,A -85,B 0,C 180,E1 15134.895,E2 15134.895} C_VEL
LIN {X 0,Y 489.557,Z 564.853,A -85,B 0,C 180,E1 15131.455,E2 15131.455} C_VEL
LIN {X 0,Y 491.409,Z 544.947,A -85,B 0,C 180,E1 15131.146,E2 15131.146} C_VEL
LIN {X 0,Y 487.605,Z 537.822,A -85,B 0,C 180,E1 15128.669,E2 15128.669} C_VEL
LIN {X 0,Y 484.467,Z 531.988,A -85,B 0,C 180,E1 15126.042,E2 15126.042} C_VEL
LIN {X 0,Y 482.057,Z 527.714,A -85,B 0,C 180,E1 15123.21,E2 15123.21} C_VEL
LIN {X 0,Y 480.279,Z 524.57,A -85,B 0,C 180,E1 15118.568,E2 15118.568} C_VEL
LIN {X 0,Y 480.35,Z 524.874,A -85,B 0,C 180,E1 15116.42,E2 15116.42} C_VEL
LIN {X 0,Y 482.425,Z 528.462,A -85,B 0,C 180,E1 15111.898,E2 15111.898} C_VEL
LIN {X 0,Y 485.072,Z 533.367,A -85,B 0,C 180,E1 15109.008,E2 15109.008} C_VEL
LIN {X 0,Y 488.432,Z 539.483,A -85,B 0,C 180,E1 15106.383,E2 15106.383} C_VEL
LIN {X 0,Y 492.342,Z 547.028,A -85,B 0,C 180,E1 15103.937,E2 15103.937} C_VEL
LIN {X 0,Y 472.159,Z 766.695,A -85,B 0,C 180,E1 15100.561,E2 15100.561} C_VEL
LIN {X 0,Y 467.367,Z 816.665,A -85,B 0,C 180,E1 15099.768,E2 15099.768} C_VEL
LIN {X 0,Y 462.94,Z 844.595,A -85,B 0,C 180,E1 15099.238,E2 15099.238} C_VEL
LIN {X 0,Y 458.241,Z 866.811,A -85,B 0,C 180,E1 15098.732,E2 15098.732} C_VEL
LIN {X 0,Y 452.744,Z 888.509,A -85,B 0,C 180,E1 15098.117,E2 15098.117} C_VEL
LIN {X 0,Y 445.181,Z 914.013,A -85,B 0,C 180,E1 15097.215,E2 15097.215} C_VEL
LIN {X 0,Y 436.734,Z 938.007,A -85,B 0,C 180,E1 15096.151,E2 15096.151} C_VEL
LIN {X 0,Y 428.861,Z 958.082,A -85,B 0,C 180,E1 15095.084,E2 15095.084} C_VEL
LIN {X 0,Y 420.445,Z 977.633,A -85,B 0,C 180,E1 15093.861,E2 15093.861} C_VEL
LIN {X 0,Y 409.454,Z 1001.023,A -85,B 0,C 180,E1 15092.126,E2 15092.126} C_VEL
LIN {X 0,Y 398.338,Z 1022.385,A -85,B 0,C 180,E1 15090.197,E2 15090.197} C_VEL
LIN {X 0,Y 388.465,Z 1040.245,A -85,B 0,C 180,E1 15088.298,E2 15088.298} C_VEL
LIN {X 0,Y 378.109,Z 1058.061,A -85,B 0,C 180,E1 15086.084,E2 15086.084} C_VEL
LIN {X 0,Y 365.327,Z 1078.889,A -85,B 0,C 180,E1 15082.977,E2 15082.977} C_VEL
LIN {X 0,Y 355.893,Z 1093.749,A -85,B 0,C 180,E1 15080.335,E2 15080.335} C_VEL
LIN {X 0,Y 347.098,Z 1107.413,A -85,B 0,C 180,E1 15077.514,E2 15077.514} C_VEL
LIN {X 0,Y 337.873,Z 1121.758,A -85,B 0,C 180,E1 15074.061,E2 15074.061} C_VEL
LIN {X 0,Y 328.057,Z 1137.236,A -85,B 0,C 180,E1 15069.568,E2 15069.568} C_VEL
LIN {X 0,Y 321.272,Z 1148.425,A -85,B 0,C 180,E1 15065.678,E2 15065.678} C_VEL
LIN {X 0,Y 316.04,Z 1157.727,A -85,B 0,C 180,E1 15061.893,E2 15061.893} C_VEL
LIN {X 0,Y 311.092,Z 1167.598,A -85,B 0,C 180,E1 15057.155,E2 15057.155} C_VEL
LIN {X 0,Y 307.519,Z 1176.033,A -85,B 0,C 180,E1 15052.078,E2 15052.078} C_VEL
LIN {X 0,Y 305.681,Z 1181.709,A -85,B 0,C 180,E1 15047.848,E2 15047.848} C_VEL
LIN {X 0,Y 304.772,Z 1185.791,A -85,B 0,C 180,E1 15044.05,E2 15044.05} C_VEL
LIN {X 0,Y 304.385,Z 1188.938,A -85,B 0,C 180,E1 15040.217,E2 15040.217} C_VEL
LIN {X 0,Y 304.326,Z 1190.999,A -85,B 0,C 180,E1 15036.603,E2 15036.603} C_VEL
LIN {X 0,Y 304.389,Z 1192.147,A -85,B 0,C 180,E1 15033.013,E2 15033.013} C_VEL
LIN {X 0,Y 304.415,Z 1192.367,A -85,B 0,C 180,E1 15029.436,E2 15029.436} C_VEL
LIN {X 0,Y 304.38,Z 1191.648,A -85,B 0,C 180,E1 15025.856,E2 15025.856} C_VEL
LIN {X 0,Y 304.359,Z 1189.86,A -85,B 0,C 180,E1 15022.069,E2 15022.069} C_VEL
LIN {X 0,Y 304.516,Z 1187.021,A -85,B 0,C 180,E1 15018.254,E2 15018.254} C_VEL
LIN {X 0,Y 305.116,Z 1183.122,A -85,B 0,C 180,E1 15014.413,E2 15014.413} C_VEL
LIN {X 0,Y 306.276,Z 1178.138,A -85,B 0,C 180,E1 15010.55,E2 15010.55} C_VEL
LIN {X 0,Y 308.22,Z 1172.051,A -85,B 0,C 180,E1 15006.686,E2 15006.686} C_VEL
LIN {X 0,Y 311.006,Z 1164.822,A -85,B 0,C 180,E1 15002.838,E2 15002.838} C_VEL
LIN {X 0,Y 315.626,Z 1154.633,A -85,B 0,C 180,E1 14998.274,E2 14998.274} C_VEL
LIN {X 0,Y 321.688,Z 1142.425,A -85,B 0,C 180,E1 14993.804,E2 14993.804} C_VEL
LIN {X 0,Y 327.92,Z 1130.76,A -85,B 0,C 180,E1 14990.185,E2 14990.185} C_VEL
LIN {X 0,Y 335.034,Z 1117.842,A -85,B 0,C 180,E1 14986.736,E2 14986.736} C_VEL
LIN {X 0,Y 344.8,Z 1100.365,A -85,B 0,C 180,E1 14982.807,E2 14982.807} C_VEL
LIN {X 0,Y 353.259,Z 1085.021,A -85,B 0,C 180,E1 14979.912,E2 14979.912} C_VEL
LIN {X 0,Y 361.434,Z 1069.922,A -85,B 0,C 180,E1 14977.444,E2 14977.444} C_VEL
LIN {X 0,Y 370.485,Z 1052.691,A -85,B 0,C 180,E1 14975.007,E2 14975.007} C_VEL
LIN {X 0,Y 381.664,Z 1030.258,A -85,B 0,C 180,E1 14972.343,E2 14972.343} C_VEL
LIN {X 0,Y 390.32,Z 1011.645,A -85,B 0,C 180,E1 14970.479,E2 14970.479} C_VEL
LIN {X 0,Y 398.464,Z 993.003,A -85,B 0,C 180,E1 14968.868,E2 14968.868} C_VEL
LIN {X 0,Y 407.224,Z 971.439,A -85,B 0,C 180,E1 14967.275,E2 14967.275} C_VEL
LIN {X 0,Y 416.271,Z 946.502,A -85,B 0,C 180,E1 14965.747,E2 14965.747} C_VEL
LIN {X 0,Y 423.174,Z 925.15,A -85,B 0,C 180,E1 14964.658,E2 14964.658} C_VEL
LIN {X 0,Y 429.304,Z 903.921,A -85,B 0,C 180,E1 14963.751,E2 14963.751} C_VEL
LIN {X 0,Y 435.848,Z 877.74,A -85,B 0,C 180,E1 14962.834,E2 14962.834} C_VEL
LIN {X 0,Y 441.023,Z 851.749,A -85,B 0,C 180,E1 14962.14,E2 14962.14} C_VEL
LIN {X 0,Y 444.511,Z 829.525,A -85,B 0,C 180,E1 14961.664,E2 14961.664} C_VEL
LIN {X 0,Y 447.206,Z 804.68,A -85,B 0,C 180,E1 14961.21,E2 14961.21} C_VEL
LIN {X 0,Y 464.457,Z 580.864,A -85,B 0,C 180,E1 14957.671,E2 14957.671} C_VEL
LIN {X 0,Y 468.208,Z 532.924,A -85,B 0,C 180,E1 14956.904,E2 14956.904} C_VEL
LIN {X 0,Y 461.62,Z 520.877,A -85,B 0,C 180,E1 14954.424,E2 14954.424} C_VEL
LIN {X 0,Y 455.407,Z 509.904,A -85,B 0,C 180,E1 14951.75,E2 14951.75} C_VEL
LIN {X 0,Y 450.049,Z 501.018,A -85,B 0,C 180,E1 14949.076,E2 14949.076} C_VEL
LIN {X 0,Y 445.248,Z 493.147,A -85,B 0,C 180,E1 14946.188,E2 14946.188} C_VEL
LIN {X 0,Y 442.287,Z 488.508,A -85,B 0,C 180,E1 14944.019,E2 14944.019} C_VEL
LIN {X 0,Y 440.224,Z 485.263,A -85,B 0,C 180,E1 14942.213,E2 14942.213} C_VEL
LIN {X 0,Y 437.561,Z 480.873,A -85,B 0,C 180,E1 14939.083,E2 14939.083} C_VEL
LIN {X 0,Y 435.457,Z 478.034,A -85,B 0,C 180,E1 14934.069,E2 14934.069} C_VEL
LIN {X 0,Y 435.521,Z 478.19,A -85,B 0,C 180,E1 14931.151,E2 14931.151} C_VEL
LIN {X 0,Y 437.867,Z 481.238,A -85,B 0,C 180,E1 14926.127,E2 14926.127} C_VEL
LIN {X 0,Y 441.131,Z 486.554,A -85,B 0,C 180,E1 14922.59,E2 14922.59} C_VEL
LIN {X 0,Y 444.921,Z 492.505,A -85,B 0,C 180,E1 14919.683,E2 14919.683} C_VEL
LIN {X 0,Y 449.369,Z 499.789,A -85,B 0,C 180,E1 14916.945,E2 14916.945} C_VEL
LIN {X 0,Y 454.177,Z 507.767,A -85,B 0,C 180,E1 14914.475,E2 14914.475} C_VEL
LIN {X 0,Y 460.515,Z 518.941,A -85,B 0,C 180,E1 14911.678,E2 14911.678} C_VEL
LIN {X 0,Y 465.08,Z 527.415,A -85,B 0,C 180,E1 14909.887,E2 14909.887} C_VEL
LIN {X 0,Y 446.626,Z 760.015,A -85,B 0,C 180,E1 14906.296,E2 14906.296} C_VEL
LIN {X 0,Y 442.969,Z 802.33,A -85,B 0,C 180,E1 14905.609,E2 14905.609} C_VEL
LIN {X 0,Y 439.176,Z 828.333,A -85,B 0,C 180,E1 14905.037,E2 14905.037} C_VEL
LIN {X 0,Y 435.293,Z 849.342,A -85,B 0,C 180,E1 14904.438,E2 14904.438} C_VEL
LIN {X 0,Y 430.262,Z 871.754,A -85,B 0,C 180,E1 14903.658,E2 14903.658} C_VEL
LIN {X 0,Y 423.238,Z 897.512,A -85,B 0,C 180,E1 14902.539,E2 14902.539} C_VEL
LIN {X 0,Y 416.742,Z 918.022,A -85,B 0,C 180,E1 14901.457,E2 14901.457} C_VEL
LIN {X 0,Y 409.438,Z 938.61,A -85,B 0,C 180,E1 14900.176,E2 14900.176} C_VEL
LIN {X 0,Y 399.86,Z 962.507,A -85,B 0,C 180,E1 14898.387,E2 14898.387} C_VEL
LIN {X 0,Y 391.811,Z 980.679,A -85,B 0,C 180,E1 14896.766,E2 14896.766} C_VEL
LIN {X 0,Y 383.48,Z 998.148,A -85,B 0,C 180,E1 14894.958,E2 14894.958} C_VEL
LIN {X 0,Y 373.084,Z 1018.409,A -85,B 0,C 180,E1 14892.482,E2 14892.482} C_VEL
LIN {X 0,Y 363.802,Z 1035.172,A -85,B 0,C 180,E1 14890.024,E2 14890.024} C_VEL
LIN {X 0,Y 355.608,Z 1049.37,A -85,B 0,C 180,E1 14887.599,E2 14887.599} C_VEL
LIN {X 0,Y 346.293,Z 1065.052,A -85,B 0,C 180,E1 14884.466,E2 14884.466} C_VEL
LIN {X 0,Y 337.501,Z 1079.214,A -85,B 0,C 180,E1 14881.029,E2 14881.029} C_VEL
LIN {X 0,Y 330.436,Z 1090.584,A -85,B 0,C 180,E1 14877.774,E2 14877.774} C_VEL
LIN {X 0,Y 323.147,Z 1102.553,A -85,B 0,C 180,E1 14873.718,E2 14873.718} C_VEL
LIN {X 0,Y 316.952,Z 1112.912,A -85,B 0,C 180,E1 14869.344,E2 14869.344} C_VEL
LIN {X 0,Y 312.837,Z 1120.331,A -85,B 0,C 180,E1 14865.573,E2 14865.573} C_VEL
LIN {X 0,Y 309.2,Z 1127.735,A -85,B 0,C 180,E1 14860.999,E2 14860.999} C_VEL
LIN {X 0,Y 306.708,Z 1133.613,A -85,B 0,C 180,E1 14856.176,E2 14856.176} C_VEL
LIN {X 0,Y 305.502,Z 1137.253,A -85,B 0,C 180,E1 14852.251,E2 14852.251} C_VEL
LIN {X 0,Y 304.915,Z 1139.792,A -85,B 0,C 180,E1 14848.497,E2 14848.497} C_VEL
LIN {X 0,Y 304.646,Z 1141.519,A -85,B 0,C 180,E1 14844.538,E2 14844.538} C_VEL
LIN {X 0,Y 304.614,Z 1142.347,A -85,B 0,C 180,E1 14840.172,E2 14840.172} C_VEL
LIN {X 0,Y 304.819,Z 1141.855,A -85,B 0,C 180,E1 14835.564,E2 14835.564} C_VEL
LIN {X 0,Y 305.342,Z 1140.356,A -85,B 0,C 180,E1 14831.48,E2 14831.48} C_VEL
LIN {X 0,Y 306.357,Z 1137.965,A -85,B 0,C 180,E1 14827.551,E2 14827.551} C_VEL
LIN {X 0,Y 308.214,Z 1134.39,A -85,B 0,C 180,E1 14823.405,E2 14823.405} C_VEL
LIN {X 0,Y 311.706,Z 1128.68,A -85,B 0,C 180,E1 14818.476,E2 14818.476} C_VEL
LIN {X 0,Y 316.323,Z 1121.727,A -85,B 0,C 180,E1 14813.99,E2 14813.99} C_VEL
LIN {X 0,Y 321.543,Z 1114.455,A -85,B 0,C 180,E1 14810.166,E2 14810.166} C_VEL
LIN {X 0,Y 329.184,Z 1104.345,A -85,B 0,C 180,E1 14805.795,E2 14805.795} C_VEL
LIN {X 0,Y 338.073,Z 1092.469,A -85,B 0,C 180,E1 14801.718,E2 14801.718} C_VEL
LIN {X 0,Y 346.419,Z 1081.376,A -85,B 0,C 180,E1 14798.539,E2 14798.539} C_VEL
LIN {X 0,Y 356.964,Z 1067.175,A -85,B 0,C 180,E1 14795.125,E2 14795.125} C_VEL
LIN {X 0,Y 361.118,Z 1061.219,A -85,B 0,C 180,E1 14793.903,E2 14793.903} C_VEL
LIN {X 0,Y 363.538,Z 1057.117,A -85,B 0,C 180,E1 14792.937,E2 14792.937} C_VEL
LIN {X 0,Y 367.583,Z 1046.498,A -85,B 0,C 180,E1 14790.123,E2 14790.123} C_VEL
LIN {X 0,Y 369.861,Z 1042.527,A -85,B 0,C 180,E1 14789.373,E2 14789.373} C_VEL
LIN {X 0,Y 380.359,Z 1026.753,A -85,B 0,C 180,E1 14787.051,E2 14787.051} C_VEL
LIN {X 0,Y 389.888,Z 1011.58,A -85,B 0,C 180,E1 14785.142,E2 14785.142} C_VEL
LIN {X 0,Y 401.109,Z 992.499,A -85,B 0,C 180,E1 14783.1,E2 14783.1} C_VEL
LIN {X 0,Y 412.024,Z 971.881,A -85,B 0,C 180,E1 14781.274,E2 14781.274} C_VEL
LIN {X 0,Y 421.031,Z 953.231,A -85,B 0,C 180,E1 14779.879,E2 14779.879} C_VEL
LIN {X 0,Y 429.765,Z 933.325,A -85,B 0,C 180,E1 14778.613,E2 14778.613} C_VEL
LIN {X 0,Y 439.329,Z 908.51,A -85,B 0,C 180,E1 14777.306,E2 14777.306} C_VEL
LIN {X 0,Y 446.269,Z 887.581,A -85,B 0,C 180,E1 14776.398,E2 14776.398} C_VEL
LIN {X 0,Y 452.097,Z 867.261,A -85,B 0,C 180,E1 14775.654,E2 14775.654} C_VEL
LIN {X 0,Y 458.3,Z 841.619,A -85,B 0,C 180,E1 14774.894,E2 14774.894} C_VEL
LIN {X 0,Y 462.978,Z 815.826,A -85,B 0,C 180,E1 14774.32,E2 14774.32} C_VEL
LIN {X 0,Y 465.928,Z 793.82,A -85,B 0,C 180,E1 14773.935,E2 14773.935} C_VEL
LIN {X 0,Y 488.179,Z 559.489,A -85,B 0,C 180,E1 14770.46,E2 14770.46} C_VEL
LIN {X 0,Y 489.001,Z 550.621,A -85,B 0,C 180,E1 14770.313,E2 14770.313} C_VEL
LIN {X 0,Y 485.613,Z 544.207,A -85,B 0,C 180,E1 14767.93,E2 14767.93} C_VEL
LIN {X 0,Y 482.989,Z 539.361,A -85,B 0,C 180,E1 14765.584,E2 14765.584} C_VEL
LIN {X 0,Y 480.995,Z 535.594,A -85,B 0,C 180,E1 14763.098,E2 14763.098} C_VEL
LIN {X 0,Y 479.299,Z 532.514,A -85,B 0,C 180,E1 14758.566,E2 14758.566} C_VEL
LIN {X 0,Y 479.37,Z 532.833,A -85,B 0,C 180,E1 14756.412,E2 14756.412} C_VEL
LIN {X 0,Y 481.311,Z 536.269,A -85,B 0,C 180,E1 14752.059,E2 14752.059} C_VEL
LIN {X 0,Y 483.882,Z 541.192,A -85,B 0,C 180,E1 14749.161,E2 14749.161} C_VEL
LIN {X 0,Y 487.094,Z 547.215,A -85,B 0,C 180,E1 14746.587,E2 14746.587} C_VEL
LIN {X 0,Y 489.858,Z 552.678,A -85,B 0,C 180,E1 14744.763,E2 14744.763} C_VEL
LIN {X 0,Y 469.524,Z 769.308,A -85,B 0,C 180,E1 14741.454,E2 14741.454} C_VEL
LIN {X 0,Y 464.787,Z 817.289,A -85,B 0,C 180,E1 14740.696,E2 14740.696} C_VEL
LIN {X 0,Y 460.297,Z 844.729,A -85,B 0,C 180,E1 14740.177,E2 14740.177} C_VEL
LIN {X 0,Y 455.56,Z 866.711,A -85,B 0,C 180,E1 14739.684,E2 14739.684} C_VEL
LIN {X 0,Y 450.074,Z 887.965,A -85,B 0,C 180,E1 14739.093,E2 14739.093} C_VEL
LIN {X 0,Y 442.522,Z 913.054,A -85,B 0,C 180,E1 14738.223,E2 14738.223} C_VEL
LIN {X 0,Y 433.909,Z 937.093,A -85,B 0,C 180,E1 14737.179,E2 14737.179} C_VEL
LIN {X 0,Y 425.876,Z 957.209,A -85,B 0,C 180,E1 14736.129,E2 14736.129} C_VEL
LIN {X 0,Y 417.58,Z 976.112,A -85,B 0,C 180,E1 14734.97,E2 14734.97} C_VEL
LIN {X 0,Y 407.096,Z 998.053,A -85,B 0,C 180,E1 14733.382,E2 14733.382} C_VEL
LIN {X 0,Y 395.179,Z 1020.61,A -85,B 0,C 180,E1 14731.397,E2 14731.397} C_VEL
LIN {X 0,Y 385.115,Z 1038.392,A -85,B 0,C 180,E1 14729.537,E2 14729.537} C_VEL
LIN {X 0,Y 375.489,Z 1054.51,A -85,B 0,C 180,E1 14727.577,E2 14727.577} C_VEL
LIN {X 0,Y 364.762,Z 1071.716,A -85,B 0,C 180,E1 14725.139,E2 14725.139} C_VEL
LIN {X 0,Y 352.175,Z 1091,A -85,B 0,C 180,E1 14721.853,E2 14721.853} C_VEL
LIN {X 0,Y 342.41,Z 1105.566,A -85,B 0,C 180,E1 14718.884,E2 14718.884} C_VEL
LIN {X 0,Y 333.566,Z 1118.685,A -85,B 0,C 180,E1 14715.758,E2 14715.758} C_VEL
LIN {X 0,Y 323.765,Z 1133.485,A -85,B 0,C 180,E1 14711.603,E2 14711.603} C_VEL
LIN {X 0,Y 315.211,Z 1146.652,A -85,B 0,C 180,E1 14707.063,E2 14707.063} C_VEL
LIN {X 0,Y 309.376,Z 1156.333,A -85,B 0,C 180,E1 14703.106,E2 14703.106} C_VEL
LIN {X 0,Y 304.738,Z 1164.769,A -85,B 0,C 180,E1 14699.051,E2 14699.051} C_VEL
LIN {X 0,Y 300.584,Z 1173.653,A -85,B 0,C 180,E1 14693.943,E2 14693.943} C_VEL
LIN {X 0,Y 297.993,Z 1180.58,A -85,B 0,C 180,E1 14688.791,E2 14688.791} C_VEL
LIN {X 0,Y 296.88,Z 1184.997,A -85,B 0,C 180,E1 14684.631,E2 14684.631} C_VEL
LIN {X 0,Y 296.417,Z 1188.181,A -85,B 0,C 180,E1 14680.692,E2 14680.692} C_VEL
LIN {X 0,Y 296.345,Z 1190.281,A -85,B 0,C 180,E1 14676.977,E2 14676.977} C_VEL
LIN {X 0,Y 296.405,Z 1191.466,A -85,B 0,C 180,E1 14673.288,E2 14673.288} C_VEL
LIN {X 0,Y 296.443,Z 1191.721,A -85,B 0,C 180,E1 14669.614,E2 14669.614} C_VEL
LIN {X 0,Y 296.406,Z 1191.034,A -85,B 0,C 180,E1 14665.938,E2 14665.938} C_VEL
LIN {X 0,Y 296.379,Z 1189.273,A -85,B 0,C 180,E1 14662.05,E2 14662.05} C_VEL
LIN {X 0,Y 296.541,Z 1186.456,A -85,B 0,C 180,E1 14658.131,E2 14658.131} C_VEL
LIN {X 0,Y 297.168,Z 1182.578,A -85,B 0,C 180,E1 14654.185,E2 14654.185} C_VEL
LIN {X 0,Y 298.391,Z 1177.617,A -85,B 0,C 180,E1 14650.219,E2 14650.219} C_VEL
LIN {X 0,Y 300.442,Z 1171.522,A -85,B 0,C 180,E1 14646.237,E2 14646.237} C_VEL
LIN {X 0,Y 303.36,Z 1164.333,A -85,B 0,C 180,E1 14642.308,E2 14642.308} C_VEL
LIN {X 0,Y 307.785,Z 1154.963,A -85,B 0,C 180,E1 14637.985,E2 14637.985} C_VEL
LIN {X 0,Y 314.545,Z 1141.995,A -85,B 0,C 180,E1 14633.074,E2 14633.074} C_VEL
LIN {X 0,Y 321.028,Z 1130.345,A -85,B 0,C 180,E1 14629.388,E2 14629.388} C_VEL
LIN {X 0,Y 328.234,Z 1117.768,A -85,B 0,C 180,E1 14625.966,E2 14625.966} C_VEL
LIN {X 0,Y 337.63,Z 1101.66,A -85,B 0,C 180,E1 14622.239,E2 14622.239} C_VEL
LIN {X 0,Y 347.298,Z 1084.689,A -85,B 0,C 180,E1 14618.984,E2 14618.984} C_VEL
LIN {X 0,Y 355.731,Z 1069.61,A -85,B 0,C 180,E1 14616.5,E2 14616.5} C_VEL
LIN {X 0,Y 364.752,Z 1052.936,A -85,B 0,C 180,E1 14614.123,E2 14614.123} C_VEL
LIN {X 0,Y 376.015,Z 1031.091,A -85,B 0,C 180,E1 14611.494,E2 14611.494} C_VEL
LIN {X 0,Y 385.271,Z 1011.733,A -85,B 0,C 180,E1 14609.545,E2 14609.545} C_VEL
LIN {X 0,Y 393.743,Z 992.812,A -85,B 0,C 180,E1 14607.908,E2 14607.908} C_VEL
LIN {X 0,Y 402.349,Z 972.146,A -85,B 0,C 180,E1 14606.381,E2 14606.381} C_VEL
LIN {X 0,Y 411.942,Z 946.439,A -85,B 0,C 180,E1 14604.802,E2 14604.802} C_VEL
LIN {X 0,Y 418.997,Z 925.097,A -85,B 0,C 180,E1 14603.719,E2 14603.719} C_VEL
LIN {X 0,Y 425.231,Z 903.957,A -85,B 0,C 180,E1 14602.821,E2 14602.821} C_VEL
LIN {X 0,Y 431.703,Z 878.714,A -85,B 0,C 180,E1 14601.938,E2 14601.938} C_VEL
LIN {X 0,Y 437.186,Z 851.926,A -85,B 0,C 180,E1 14601.223,E2 14601.223} C_VEL
LIN {X 0,Y 440.764,Z 829.644,A -85,B 0,C 180,E1 14600.748,E2 14600.748} C_VEL
LIN {X 0,Y 443.434,Z 805.836,A -85,B 0,C 180,E1 14600.312,E2 14600.312} C_VEL
LIN {X 0,Y 460.946,Z 584.437,A -85,B 0,C 180,E1 14596.817,E2 14596.817} C_VEL
LIN {X 0,Y 464.654,Z 537.525,A -85,B 0,C 180,E1 14596.053,E2 14596.053} C_VEL
LIN {X 0,Y 458.02,Z 525.158,A -85,B 0,C 180,E1 14593.412,E2 14593.412} C_VEL
LIN {X 0,Y 451.746,Z 514.037,A -85,B 0,C 180,E1 14590.522,E2 14590.522} C_VEL
LIN {X 0,Y 446.711,Z 505.591,A -85,B 0,C 180,E1 14587.783,E2 14587.783} C_VEL
LIN {X 0,Y 443.122,Z 499.659,A -85,B 0,C 180,E1 14585.438,E2 14585.438} C_VEL
LIN {X 0,Y 439.582,Z 493.724,A -85,B 0,C 180,E1 14582.542,E2 14582.542} C_VEL
LIN {X 0,Y 436.477,Z 488.746,A -85,B 0,C 180,E1 14578.95,E2 14578.95} C_VEL
LIN {X 0,Y 434.461,Z 485.94,A -85,B 0,C 180,E1 14573.923,E2 14573.923} C_VEL
LIN {X 0,Y 434.567,Z 486.203,A -85,B 0,C 180,E1 14570.998,E2 14570.998} C_VEL
LIN {X 0,Y 436.797,Z 489.172,A -85,B 0,C 180,E1 14566.227,E2 14566.227} C_VEL
LIN {X 0,Y 439.875,Z 494.272,A -85,B 0,C 180,E1 14562.812,E2 14562.812} C_VEL
LIN {X 0,Y 443.769,Z 500.504,A -85,B 0,C 180,E1 14559.765,E2 14559.765} C_VEL
LIN {X 0,Y 448.171,Z 507.952,A -85,B 0,C 180,E1 14557.018,E2 14557.018} C_VEL
LIN {X 0,Y 453.339,Z 516.762,A -85,B 0,C 180,E1 14554.351,E2 14554.351} C_VEL
LIN {X 0,Y 460.04,Z 528.988,A -85,B 0,C 180,E1 14551.402,E2 14551.402} C_VEL
LIN {X 0,Y 461.686,Z 532.329,A -85,B 0,C 180,E1 14550.733,E2 14550.733} C_VEL
LIN {X 0,Y 442.817,Z 764.643,A -85,B 0,C 180,E1 14547.158,E2 14547.158} C_VEL
LIN {X 0,Y 439.294,Z 803.572,A -85,B 0,C 180,E1 14546.522,E2 14546.522} C_VEL
LIN {X 0,Y 435.499,Z 829.004,A -85,B 0,C 180,E1 14545.964,E2 14545.964} C_VEL
LIN {X 0,Y 431.533,Z 849.995,A -85,B 0,C 180,E1 14545.368,E2 14545.368} C_VEL
LIN {X 0,Y 426.338,Z 872.636,A -85,B 0,C 180,E1 14544.584,E2 14544.584} C_VEL
LIN {X 0,Y 419.251,Z 898.027,A -85,B 0,C 180,E1 14543.485,E2 14543.485} C_VEL
LIN {X 0,Y 412.618,Z 918.534,A -85,B 0,C 180,E1 14542.409,E2 14542.409} C_VEL
LIN {X 0,Y 405.156,Z 939.126,A -85,B 0,C 180,E1 14541.133,E2 14541.133} C_VEL
LIN {X 0,Y 395.357,Z 963.037,A -85,B 0,C 180,E1 14539.35,E2 14539.35} C_VEL
LIN {X 0,Y 387.111,Z 981.216,A -85,B 0,C 180,E1 14537.731,E2 14537.731} C_VEL
LIN {X 0,Y 378.851,Z 998.111,A -85,B 0,C 180,E1 14535.986,E2 14535.986} C_VEL
LIN {X 0,Y 368.434,Z 1017.992,A -85,B 0,C 180,E1 14533.575,E2 14533.575} C_VEL
LIN {X 0,Y 358.327,Z 1035.733,A -85,B 0,C 180,E1 14530.975,E2 14530.975} C_VEL
LIN {X 0,Y 349.874,Z 1049.942,A -85,B 0,C 180,E1 14528.535,E2 14528.535} C_VEL
LIN {X 0,Y 340.24,Z 1065.629,A -85,B 0,C 180,E1 14525.374,E2 14525.374} C_VEL
LIN {X 0,Y 331.121,Z 1079.799,A -85,B 0,C 180,E1 14521.899,E2 14521.899} C_VEL
LIN {X 0,Y 323.774,Z 1091.182,A -85,B 0,C 180,E1 14518.598,E2 14518.598} C_VEL
LIN {X 0,Y 316.175,Z 1103.156,A -85,B 0,C 180,E1 14514.473,E2 14514.473} C_VEL
LIN {X 0,Y 309.687,Z 1113.521,A -85,B 0,C 180,E1 14510.013,E2 14510.013} C_VEL
LIN {X 0,Y 305.36,Z 1120.947,A -85,B 0,C 180,E1 14506.16,E2 14506.16} C_VEL
LIN {X 0,Y 301.521,Z 1128.357,A -85,B 0,C 180,E1 14501.476,E2 14501.476} C_VEL
LIN {X 0,Y 298.872,Z 1134.243,A -85,B 0,C 180,E1 14496.531,E2 14496.531} C_VEL
LIN {X 0,Y 297.591,Z 1137.886,A -85,B 0,C 180,E1 14492.503,E2 14492.503} C_VEL
LIN {X 0,Y 296.961,Z 1140.431,A -85,B 0,C 180,E1 14488.649,E2 14488.649} C_VEL
LIN {X 0,Y 296.674,Z 1142.164,A -85,B 0,C 180,E1 14484.585,E2 14484.585} C_VEL
LIN {X 0,Y 296.642,Z 1143.003,A -85,B 0,C 180,E1 14480.102,E2 14480.102} C_VEL
LIN {X 0,Y 296.869,Z 1142.531,A -85,B 0,C 180,E1 14475.368,E2 14475.368} C_VEL
LIN {X 0,Y 297.438,Z 1141.046,A -85,B 0,C 180,E1 14471.173,E2 14471.173} C_VEL
LIN {X 0,Y 298.562,Z 1138.622,A -85,B 0,C 180,E1 14467.071,E2 14467.071} C_VEL
